C03633=1108.263,416.808,-95.419,-178.655,16.482,151.225
C03634=1108.269,417.055,-95.459,-178.654,16.489,151.227
C03635=1108.274,417.302,-95.498,-178.652,16.496,151.228
C03636=1108.279,417.549,-95.536,-178.650,16.503,151.230
C03637=1108.285,417.796,-95.575,-178.649,16.510,151.231
C03638=1108.291,418.042,-95.614,-178.647,16.517,151.232
C03639=1108.297,418.289,-95.654,-178.645,16.524,151.234
C03640=1108.302,418.536,-95.693,-178.644,16.531,151.235
C03641=1108.307,418.783,-95.733,-178.642,16.538,151.237
C03642=1108.313,419.030,-95.772,-178.640,16.545,151.238
C03643=1108.319,419.276,-95.811,-178.639,16.553,151.240
C03644=1108.325,419.523,-95.851,-178.638,16.560,151.241
C03645=1108.330,419.770,-95.890,-178.636,16.567,151.243
C03646=1108.336,420.017,-95.929,-178.634,16.574,151.244
C03647=1108.342,420.264,-95.967,-178.632,16.582,151.246
C03648=1108.347,420.510,-96.008,-178.631,16.589,151.247
C03649=1108.353,420.757,-96.047,-178.629,16.596,151.249
C03650=1108.358,421.004,-96.086,-178.627,16.603,151.250
C03651=1108.364,421.251,-96.126,-178.626,16.611,151.252
C03652=1108.370,421.497,-96.165,-178.625,16.618,151.254
C03653=1108.375,421.745,-96.205,-178.623,16.625,151.255
C03654=1108.381,421.991,-96.244,-178.621,16.633,151.257
C03655=1108.387,422.238,-96.283,-178.619,16.640,151.258
C03656=1108.392,422.485,-96.322,-178.618,16.648,151.260
C03657=1108.398,422.732,-96.362,-178.616,16.655,151.261
C03658=1108.403,422.978,-96.402,-178.615,16.663,151.263
C03659=1108.409,423.225,-96.442,-178.614,16.670,151.265
C03660=1108.414,423.443,-96.476,-178.612,16.678,151.266
C03661=1108.419,423.661,-96.511,-178.611,16.684,151.268
C03662=1108.424,423.879,-96.546,-178.610,16.691,151.269
C03663=1108.429,424.099,-96.582,-178.608,16.698,151.271
C03664=1108.434,424.317,-96.617,-178.607,16.704,151.272
C03665=1108.439,424.535,-96.652,-178.606,16.712,151.274
C03666=1108.443,424.753,-96.687,-178.604,16.718,151.275
C03667=1108.449,424.972,-96.722,-178.603,16.725,151.277
C03668=1108.454,425.218,-96.762,-178.602,16.733,151.278
C03669=1108.460,425.465,-96.802,-178.600,16.741,151.280
C03670=1108.465,425.712,-96.842,-178.599,16.749,151.282
C03671=1108.471,425.959,-96.881,-178.598,16.757,151.283
C03672=1108.477,426.205,-96.921,-178.596,16.764,151.285
C03673=1108.482,426.452,-96.961,-178.595,16.773,151.287
C03674=1108.488,426.698,-97.001,-178.593,16.781,151.289
C03675=1108.493,426.945,-97.041,-178.592,16.789,151.290
C03676=1108.500,427.192,-97.081,-178.591,16.797,151.292
C03677=1108.504,427.439,-97.121,-178.589,16.805,151.294
C03678=1108.511,427.685,-97.161,-178.588,16.813,151.296
C03679=1108.515,427.932,-97.200,-178.587,16.821,151.298
C03680=1108.522,428.178,-97.240,-178.585,16.829,151.299
C03681=1108.527,428.426,-97.281,-178.584,16.837,151.301
C03682=1108.533,428.672,-97.320,-178.583,16.845,151.303
C03683=1108.539,428.918,-97.361,-178.582,16.854,151.305
C03684=1108.544,429.165,-97.400,-178.580,16.862,151.307
C03685=1108.550,429.412,-97.441,-178.579,16.870,151.309
C03686=1108.556,429.659,-97.480,-178.578,16.879,151.311
C03687=1108.561,429.905,-97.521,-178.577,16.887,151.312
C03688=1108.566,430.152,-97.561,-178.575,16.896,151.314
C03689=1108.572,430.398,-97.601,-178.574,16.904,151.316
C03690=1108.578,430.645,-97.641,-178.573,16.913,151.318
C03691=1108.584,430.892,-97.681,-178.572,16.921,151.320
C03692=1108.589,431.138,-97.722,-178.571,16.930,151.322
C03693=1108.595,431.384,-97.762,-178.570,16.938,151.324
C03694=1108.601,431.632,-97.802,-178.568,16.946,151.326
C03695=1108.606,431.878,-97.842,-178.567,16.956,151.328
C03696=1108.611,432.125,-97.883,-178.566,16.964,151.330
C03697=1108.617,432.371,-97.924,-178.565,16.973,151.332
C03698=1108.623,432.617,-97.964,-178.564,16.981,151.334
C03699=1108.628,432.864,-98.004,-178.563,16.990,151.336
C03700=1108.634,433.111,-98.044,-178.561,16.999,151.338
C03701=1108.640,433.357,-98.084,-178.560,17.008,151.340
C03702=1108.645,433.604,-98.125,-178.560,17.017,151.342
C03703=1108.651,433.851,-98.166,-178.559,17.025,151.344
C03704=1108.656,434.097,-98.206,-178.558,17.034,151.346
C03705=1108.662,434.344,-98.247,-178.556,17.044,151.348
C03706=1108.667,434.591,-98.287,-178.556,17.052,151.351
C03707=1108.673,434.837,-98.327,-178.555,17.061,151.353
C03708=1108.679,435.083,-98.368,-178.553,17.071,151.355
C03709=1108.684,435.330,-98.409,-178.553,17.080,151.357
C03710=1108.689,435.576,-98.449,-178.552,17.089,151.359
C03711=1108.695,435.823,-98.490,-178.551,17.098,151.361
C03712=1108.701,436.069,-98.531,-178.550,17.107,151.364
C03713=1108.706,436.315,-98.572,-178.549,17.117,151.366
C03714=1108.712,436.562,-98.612,-178.549,17.126,151.368
C03715=1108.717,436.809,-98.653,-178.547,17.135,151.370
C03716=1108.723,437.037,-98.690,-178.546,17.144,151.372
C03717=1108.727,437.265,-98.728,-178.545,17.153,151.374
C03718=1108.733,437.493,-98.766,-178.545,17.161,151.376
C03719=1108.738,437.721,-98.804,-178.545,17.170,151.379
C03720=1108.743,437.949,-98.841,-178.544,17.179,151.381
C03721=1108.749,438.177,-98.879,-178.543,17.188,151.383
C03722=1108.754,438.406,-98.917,-178.542,17.196,151.385
C03723=1108.758,438.634,-98.954,-178.541,17.205,151.387
C03724=1108.764,438.880,-98.996,-178.541,17.215,151.389
C03725=1108.770,439.127,-99.037,-178.540,17.224,151.392
C03726=1108.776,439.373,-99.078,-178.539,17.234,151.394
C03727=1108.782,439.620,-99.119,-178.538,17.244,151.396
C03728=1108.787,439.866,-99.159,-178.538,17.254,151.399
C03729=1108.793,440.112,-99.201,-178.537,17.264,151.401
C03730=1108.798,440.359,-99.241,-178.536,17.273,151.403
C03731=1108.804,440.606,-99.282,-178.536,17.283,151.406
C03732=1108.810,440.852,-99.324,-178.535,17.293,151.408
C03733=1108.815,441.098,-99.364,-178.535,17.303,151.411
C03734=1108.821,441.345,-99.405,-178.534,17.313,151.413
C03735=1108.826,441.591,-99.446,-178.534,17.323,151.416
C03736=1108.832,441.838,-99.488,-178.533,17.333,151.418
C03737=1108.838,442.084,-99.530,-178.532,17.343,151.420
C03738=1108.843,442.330,-99.570,-178.532,17.353,151.423
C03739=1108.849,442.576,-99.611,-178.531,17.364,151.426
C03740=1108.854,442.823,-99.652,-178.530,17.374,151.428
C03741=1108.860,443.069,-99.694,-178.530,17.384,151.431
C03742=1108.865,443.317,-99.735,-178.530,17.394,151.433
C03743=1108.871,443.563,-99.776,-178.529,17.405,151.436
C03744=1108.876,443.808,-99.818,-178.529,17.415,151.438
C03745=1108.881,444.055,-99.859,-178.529,17.425,151.441
C03746=1108.887,444.302,-99.900,-178.529,17.435,151.444
C03747=1108.893,444.548,-99.942,-178.529,17.445,151.446
C03748=1108.899,444.795,-99.983,-178.530,17.456,151.449
C03749=1108.904,445.041,-100.025,-178.530,17.466,151.452
C03750=1108.910,445.287,-100.066,-178.530,17.477,151.454
C03751=1108.916,445.534,-100.108,-178.531,17.486,151.457
C03752=1108.921,445.781,-100.149,-178.531,17.497,151.460
C03753=1108.926,446.026,-100.190,-178.532,17.506,151.463
C03754=1108.932,446.272,-100.231,-178.533,17.517,151.465
C03755=1108.937,446.519,-100.273,-178.534,17.527,151.468
C03756=1108.943,446.766,-100.314,-178.535,17.537,151.471
C03757=1108.948,447.012,-100.356,-178.537,17.547,151.474
C03758=1108.954,447.259,-100.398,-178.538,17.557,151.477
C03759=1108.959,447.505,-100.440,-178.539,17.567,151.480
C03760=1108.965,447.751,-100.481,-178.540,17.577,151.482
C03761=1108.970,447.998,-100.523,-178.541,17.587,151.485
C03762=1108.976,448.245,-100.564,-178.544,17.597,151.488
C03763=1108.981,448.491,-100.606,-178.545,17.608,151.491
C03764=1108.987,448.737,-100.648,-178.547,17.617,151.494
C03765=1108.993,448.983,-100.689,-178.549,17.628,151.497
C03766=1108.998,449.230,-100.731,-178.551,17.637,151.500
C03767=1109.004,449.476,-100.772,-178.553,17.647,151.503
C03768=1109.010,449.723,-100.815,-178.555,17.658,151.506
C03769=1109.016,449.969,-100.856,-178.557,17.667,151.509
C03770=1109.020,450.216,-100.897,-178.559,17.677,151.512
C03771=1109.026,450.462,-100.939,-178.561,17.687,151.515
C03772=1108.617,450.455,-101.049,-178.646,17.920,151.591
C03773=1108.612,450.209,-101.007,-178.644,17.910,151.588
C03774=1108.606,449.963,-100.965,-178.642,17.900,151.585
C03775=1108.600,449.716,-100.923,-178.640,17.890,151.582
C03776=1108.594,449.470,-100.882,-178.638,17.880,151.579
C03777=1108.589,449.223,-100.840,-178.635,17.870,151.576
C03778=1108.583,448.977,-100.798,-178.634,17.859,151.573
C03779=1108.578,448.731,-100.756,-178.632,17.850,151.570
C03780=1108.572,448.484,-100.715,-178.631,17.839,151.568
C03781=1108.567,448.238,-100.673,-178.628,17.830,151.565
C03782=1108.561,447.992,-100.631,-178.627,17.819,151.562
C03783=1108.556,447.745,-100.589,-178.626,17.809,151.559
C03784=1108.550,447.498,-100.548,-178.624,17.799,151.556
C03785=1108.545,447.252,-100.506,-178.622,17.789,151.553
C03786=1108.539,447.006,-100.465,-178.621,17.779,151.550
C03787=1108.534,446.759,-100.423,-178.620,17.769,151.547
C03788=1108.528,446.513,-100.381,-178.620,17.758,151.544
C03789=1108.523,446.266,-100.339,-178.618,17.748,151.542
C03790=1108.517,446.020,-100.298,-178.617,17.738,151.539
C03791=1108.511,445.773,-100.257,-178.617,17.727,151.536
C03792=1108.506,445.528,-100.215,-178.616,17.717,151.533
C03793=1108.500,445.281,-100.174,-178.616,17.707,151.530
C03794=1108.495,445.035,-100.133,-178.615,17.696,151.528
C03795=1108.489,444.789,-100.090,-178.615,17.687,151.525
C03796=1108.484,444.542,-100.050,-178.614,17.676,151.522
C03797=1108.478,444.296,-100.008,-178.614,17.666,151.520
C03798=1108.472,444.049,-99.966,-178.614,17.656,151.517
C03799=1108.467,443.803,-99.925,-178.615,17.645,151.515
C03800=1108.461,443.556,-99.884,-178.615,17.635,151.512
C03801=1108.456,443.310,-99.842,-178.616,17.624,151.509
C03802=1108.450,443.064,-99.801,-178.616,17.614,151.507
C03803=1108.445,442.817,-99.760,-178.617,17.603,151.504
C03804=1108.439,442.571,-99.719,-178.617,17.593,151.502
C03805=1108.434,442.325,-99.677,-178.618,17.583,151.499
C03806=1108.428,442.078,-99.636,-178.618,17.573,151.497
C03807=1108.422,441.832,-99.594,-178.619,17.563,151.494
C03808=1108.417,441.585,-99.554,-178.620,17.552,151.492
C03809=1108.411,441.339,-99.513,-178.620,17.542,151.489
C03810=1108.405,441.092,-99.472,-178.621,17.532,151.487
C03811=1108.400,440.846,-99.430,-178.621,17.522,151.484
C03812=1108.394,440.600,-99.388,-178.622,17.511,151.482
C03813=1108.389,440.353,-99.348,-178.623,17.502,151.479
C03814=1108.383,440.106,-99.307,-178.624,17.492,151.477
C03815=1108.378,439.861,-99.266,-178.624,17.482,151.475
C03816=1108.372,439.614,-99.225,-178.625,17.472,151.472
C03817=1108.366,439.368,-99.184,-178.626,17.462,151.470
C03818=1108.360,439.121,-99.143,-178.626,17.453,151.467
C03819=1108.354,438.874,-99.101,-178.628,17.443,151.465
C03820=1108.349,438.628,-99.061,-178.628,17.433,151.463
C03821=1108.344,438.401,-99.023,-178.629,17.425,151.461
C03822=1108.339,438.174,-98.986,-178.630,17.416,151.459
C03823=1108.333,437.948,-98.948,-178.631,17.407,151.456
C03824=1108.328,437.721,-98.910,-178.631,17.398,151.454
C03825=1108.323,437.494,-98.873,-178.632,17.389,151.452
C03826=1108.318,437.267,-98.835,-178.633,17.380,151.450
C03827=1108.313,437.041,-98.798,-178.634,17.371,151.448
C03828=1108.308,436.815,-98.760,-178.634,17.363,151.446
C03829=1108.302,436.568,-98.719,-178.636,17.354,151.444
C03830=1108.297,436.321,-98.679,-178.636,17.344,151.442
C03831=1108.291,436.074,-98.638,-178.637,17.335,151.439
C03832=1108.286,435.828,-98.597,-178.639,17.326,151.437
C03833=1108.280,435.581,-98.557,-178.639,17.316,151.435
C03834=1108.274,435.335,-98.516,-178.640,17.308,151.433
C03835=1108.269,435.089,-98.476,-178.641,17.298,151.431
C03836=1108.263,434.843,-98.435,-178.642,17.289,151.428
C03837=1108.257,434.596,-98.394,-178.643,17.280,151.426
C03838=1108.252,434.350,-98.354,-178.644,17.270,151.424
C03839=1108.247,434.103,-98.313,-178.645,17.261,151.422
C03840=1108.241,433.856,-98.272,-178.646,17.252,151.420
C03841=1108.236,433.610,-98.232,-178.648,17.243,151.418
C03842=1108.230,433.363,-98.192,-178.649,17.234,151.416
C03843=1108.224,433.116,-98.151,-178.650,17.225,151.414
C03844=1108.218,432.870,-98.110,-178.650,17.217,151.412
C03845=1108.213,432.623,-98.070,-178.651,17.208,151.410
C03846=1108.207,432.377,-98.030,-178.653,17.198,151.408
C03847=1108.201,432.130,-97.989,-178.654,17.190,151.406
C03848=1108.196,431.883,-97.949,-178.655,17.181,151.404
C03849=1108.190,431.637,-97.909,-178.656,17.173,151.402
C03850=1108.184,431.390,-97.868,-178.657,17.164,151.400
C03851=1108.179,431.144,-97.828,-178.659,17.155,151.398
C03852=1108.173,430.897,-97.788,-178.660,17.146,151.396
C03853=1108.167,430.651,-97.747,-178.661,17.138,151.394
C03854=1108.163,430.404,-97.707,-178.662,17.129,151.392
C03855=1108.156,430.157,-97.667,-178.663,17.121,151.390
C03856=1108.151,429.911,-97.627,-178.665,17.113,151.388
C03857=1108.146,429.664,-97.587,-178.667,17.104,151.386
C03858=1108.139,429.417,-97.547,-178.668,17.095,151.384
C03859=1108.134,429.171,-97.506,-178.669,17.087,151.382
C03860=1108.128,428.925,-97.466,-178.670,17.078,151.380
C03861=1108.123,428.677,-97.426,-178.671,17.070,151.378
C03862=1108.118,428.431,-97.386,-178.673,17.062,151.377
C03863=1108.112,428.184,-97.346,-178.674,17.054,151.375
C03864=1108.106,427.937,-97.306,-178.675,17.046,151.373
C03865=1108.100,427.691,-97.266,-178.677,17.037,151.371
C03866=1108.095,427.444,-97.226,-178.678,17.029,151.369
C03867=1108.089,427.198,-97.186,-178.679,17.021,151.367
C03868=1108.083,426.951,-97.147,-178.681,17.013,151.366
C03869=1108.077,426.704,-97.106,-178.682,17.005,151.364
C03870=1108.072,426.458,-97.067,-178.684,16.997,151.362
C03871=1108.066,426.211,-97.026,-178.685,16.989,151.360
C03872=1108.061,425.964,-96.987,-178.686,16.981,151.359
C03873=1108.055,425.718,-96.946,-178.688,16.973,151.357
C03874=1108.050,425.471,-96.907,-178.689,16.965,151.355
C03875=1108.044,425.224,-96.867,-178.691,16.957,151.353
C03876=1108.039,424.978,-96.827,-178.692,16.949,151.352
C03877=1108.033,424.759,-96.793,-178.693,16.942,151.350
C03878=1108.029,424.540,-96.757,-178.695,16.935,151.349
C03879=1108.023,424.322,-96.721,-178.696,16.928,151.347
C03880=1108.019,424.103,-96.687,-178.697,16.921,151.346
C03881=1108.013,423.885,-96.652,-178.699,16.914,151.344
C03882=1108.009,423.666,-96.616,-178.700,16.907,151.343
C03883=1108.004,423.448,-96.581,-178.702,16.901,151.341
C03884=1107.999,423.230,-96.546,-178.703,16.894,151.340
C03885=1107.993,422.983,-96.506,-178.704,16.886,151.338
C03886=1107.988,422.736,-96.467,-178.706,16.878,151.336
C03887=1107.982,422.489,-96.427,-178.708,16.871,151.335
C03888=1107.976,422.243,-96.387,-178.709,16.863,151.333
C03889=1107.970,421.996,-96.348,-178.711,16.855,151.332
C03890=1107.965,421.750,-96.309,-178.712,16.848,151.330
C03891=1107.959,421.502,-96.269,-178.714,16.841,151.329
C03892=1107.954,421.256,-96.230,-178.715,16.833,151.327
C03893=1107.948,421.009,-96.190,-178.717,16.826,151.325
C03894=1107.942,420.762,-96.151,-178.719,16.818,151.324
C03895=1107.936,420.515,-96.112,-178.720,16.811,151.322
C03896=1107.931,420.268,-96.072,-178.722,16.804,151.321
C03897=1107.925,420.021,-96.033,-178.724,16.796,151.319
C03898=1107.920,419.775,-95.993,-178.725,16.789,151.318
C03899=1107.914,419.528,-95.954,-178.727,16.782,151.316
C03900=1107.908,419.282,-95.915,-178.728,16.775,151.315
C03901=1107.902,419.034,-95.876,-178.730,16.767,151.313
C03902=1107.898,418.787,-95.836,-178.732,16.760,151.312
C03903=1107.891,418.540,-95.797,-178.734,16.753,151.310
C03904=1107.886,418.294,-95.758,-178.735,16.746,151.309
C03905=1107.881,418.047,-95.719,-178.737,16.738,151.307
C03906=1107.874,417.800,-95.679,-178.739,16.731,151.306
C03907=1107.869,417.554,-95.640,-178.740,16.725,151.304
C03908=1107.863,417.307,-95.601,-178.742,16.717,151.303
C03909=1107.857,417.060,-95.562,-178.744,16.710,151.302
C03910=1107.853,416.813,-95.523,-178.746,16.703,151.300
C03911=1107.847,416.566,-95.483,-178.747,16.696,151.299
C03912=1107.841,416.320,-95.445,-178.749,16.689,151.297
C03913=1107.835,416.072,-95.405,-178.751,16.683,151.296
C03914=1107.829,415.826,-95.366,-178.753,16.676,151.294
C03915=1107.823,415.578,-95.328,-178.755,16.669,151.293
C03916=1107.818,415.332,-95.288,-178.756,16.662,151.292
C03917=1107.812,415.085,-95.249,-178.758,16.655,151.290
C03918=1107.807,414.838,-95.211,-178.760,16.649,151.289
C03919=1107.801,414.591,-95.172,-178.762,16.642,151.288
C03920=1107.795,414.344,-95.132,-178.764,16.635,151.286
C03921=1107.790,414.097,-95.094,-178.765,16.628,151.285
C03922=1107.785,413.851,-95.055,-178.768,16.621,151.284
C03923=1107.778,413.604,-95.016,-178.769,16.615,151.282
C03924=1107.773,413.357,-94.978,-178.771,16.608,151.281
C03925=1107.767,413.110,-94.939,-178.773,16.602,151.280
C03926=1107.761,412.863,-94.900,-178.775,16.595,151.279
C03927=1107.756,412.616,-94.861,-178.776,16.589,151.277
C03928=1107.751,412.369,-94.822,-178.779,16.582,151.276
C03929=1107.745,412.122,-94.783,-178.780,16.576,151.275
C03930=1107.739,411.875,-94.745,-178.782,16.569,151.273
C03931=1107.733,411.629,-94.706,-178.784,16.563,151.272
C03932=1107.727,411.381,-94.667,-178.786,16.556,151.271
C03933=1107.723,411.169,-94.634,-178.788,16.550,151.270
C03934=1107.717,410.957,-94.601,-178.789,16.545,151.269
C03935=1107.713,410.746,-94.568,-178.791,16.539,151.268
C03936=1107.708,410.534,-94.535,-178.793,16.534,151.267
C03937=1107.703,410.322,-94.502,-178.794,16.529,151.266
C03938=1107.699,410.109,-94.469,-178.796,16.523,151.265
C03939=1107.694,409.897,-94.436,-178.798,16.517,151.264
C03940=1107.689,409.686,-94.402,-178.799,16.512,151.263
C03941=1107.683,409.439,-94.364,-178.802,16.506,151.261
C03942=1107.677,409.191,-94.325,-178.803,16.500,151.260
C03943=1107.672,408.945,-94.286,-178.805,16.494,151.259
C03944=1107.667,408.698,-94.248,-178.807,16.487,151.258
C03945=1107.661,408.451,-94.210,-178.809,16.481,151.257
C03946=1107.656,408.204,-94.172,-178.811,16.474,151.256
C03947=1107.650,407.956,-94.133,-178.813,16.468,151.254
C03948=1107.644,407.710,-94.095,-178.815,16.463,151.253
C03949=1107.639,407.463,-94.056,-178.817,16.456,151.252
C03950=1107.633,407.216,-94.018,-178.819,16.450,151.251
C03951=1107.627,406.968,-93.980,-178.821,16.444,151.250
C03952=1107.622,406.721,-93.941,-178.823,16.438,151.249
C03953=1107.616,406.475,-93.902,-178.825,16.432,151.248
C03954=1107.610,406.228,-93.865,-178.827,16.426,151.247
C03955=1107.605,405.981,-93.826,-178.829,16.420,151.245
C03956=1107.599,405.734,-93.788,-178.831,16.414,151.244
C03957=1107.594,405.487,-93.750,-178.833,16.408,151.243
C03958=1107.588,405.240,-93.712,-178.835,16.402,151.242
C03959=1107.582,404.993,-93.674,-178.838,16.396,151.241
C03960=1107.577,404.746,-93.636,-178.839,16.391,151.240
C03961=1107.571,404.498,-93.597,-178.841,16.385,151.239
C03962=1107.565,404.252,-93.559,-178.843,16.379,151.238
C03963=1107.560,404.005,-93.521,-178.846,16.373,151.237
C03964=1107.554,403.758,-93.483,-178.848,16.367,151.236
C03965=1107.549,403.511,-93.445,-178.850,16.362,151.235
C03966=1107.542,403.263,-93.407,-178.852,16.356,151.234
C03967=1107.536,403.017,-93.369,-178.854,16.351,151.233
C03968=1107.531,402.769,-93.331,-178.856,16.345,151.232
C03969=1107.525,402.523,-93.293,-178.859,16.339,151.231
C03970=1107.520,402.275,-93.255,-178.860,16.333,151.230
C03971=1107.514,402.028,-93.218,-178.863,16.328,151.229
C03972=1107.509,401.782,-93.180,-178.865,16.322,151.228
C03973=1107.503,401.535,-93.142,-178.867,16.317,151.227
C03974=1107.497,401.287,-93.103,-178.869,16.311,151.226
C03975=1107.492,401.040,-93.065,-178.871,16.305,151.225
C03976=1107.486,400.793,-93.028,-178.874,16.300,151.224
C03977=1107.480,400.546,-92.990,-178.876,16.294,151.223
C03978=1107.475,400.299,-92.952,-178.878,16.289,151.223
C03979=1107.469,400.052,-92.914,-178.880,16.284,151.222
C03980=1107.464,399.805,-92.877,-178.882,16.278,151.221
C03981=1107.458,399.558,-92.839,-178.884,16.273,151.220
C03982=1107.452,399.311,-92.801,-178.886,16.267,151.219
C03983=1107.447,399.064,-92.764,-178.888,16.262,151.218
C03984=1107.441,398.817,-92.726,-178.890,16.257,151.217
C03985=1107.435,398.570,-92.688,-178.893,16.251,151.216
C03986=1107.430,398.322,-92.651,-178.895,16.246,151.215
C03987=1107.424,398.076,-92.613,-178.897,16.241,151.214
C03988=1107.418,397.829,-92.575,-178.899,16.235,151.214
C03989=1107.414,397.616,-92.543,-178.902,16.231,151.213
C03990=1107.408,397.404,-92.511,-178.903,16.226,151.212
C03991=1107.404,397.192,-92.478,-178.905,16.222,151.211
C03992=1107.398,396.979,-92.447,-178.907,16.217,151.211
C03993=1107.394,396.768,-92.414,-178.909,16.213,151.210
C03994=1107.389,396.555,-92.382,-178.911,16.208,151.209
C03995=1107.384,396.343,-92.350,-178.913,16.204,151.209
C03996=1107.380,396.131,-92.317,-178.915,16.199,151.208
C03997=1107.374,395.884,-92.280,-178.917,16.194,151.207
C03998=1107.368,395.637,-92.243,-178.920,16.189,151.206
C03999=1107.363,395.390,-92.206,-178.922,16.184,151.205
C04000=1107.357,395.143,-92.168,-178.924,16.179,151.205
C04001=1107.351,394.896,-92.131,-178.927,16.174,151.204
C04002=1107.346,394.648,-92.094,-178.929,16.168,151.203
C04003=1107.340,394.401,-92.056,-178.931,16.164,151.202
C04004=1107.334,394.154,-92.019,-178.934,16.159,151.202
C04005=1107.328,393.907,-91.981,-178.936,16.153,151.201
C04006=1107.323,393.660,-91.944,-178.938,16.149,151.200
C04007=1107.317,393.413,-91.907,-178.940,16.144,151.199
C04008=1107.311,393.166,-91.869,-178.943,16.139,151.198
C04009=1107.306,392.919,-91.832,-178.945,16.134,151.198
C04010=1107.300,392.671,-91.795,-178.948,16.129,151.197
C04011=1107.294,392.424,-91.758,-178.950,16.124,151.196
C04012=1107.289,392.178,-91.721,-178.953,16.119,151.196
C04013=1107.283,391.930,-91.684,-178.955,16.115,151.195
C04014=1107.278,391.683,-91.647,-178.958,16.110,151.194
C04015=1107.272,391.436,-91.610,-178.960,16.105,151.193
C04016=1107.266,391.189,-91.573,-178.962,16.101,151.193
C04017=1107.260,390.942,-91.536,-178.964,16.096,151.192
C04018=1107.254,390.695,-91.499,-178.967,16.091,151.191
C04019=1107.249,390.447,-91.462,-178.969,16.086,151.191
C04020=1107.243,390.200,-91.424,-178.972,16.081,151.190
C04021=1107.238,389.954,-91.387,-178.975,16.076,151.189
C04022=1107.232,389.707,-91.351,-178.977,16.072,151.189
C04023=1107.226,389.459,-91.314,-178.979,16.067,151.188
C04024=1107.220,389.212,-91.277,-178.981,16.062,151.187
C04025=1107.215,388.965,-91.240,-178.984,16.058,151.187
C04026=1107.208,388.718,-91.203,-178.987,16.053,151.186
C04027=1107.203,388.471,-91.166,-178.989,16.048,151.186
C04028=1107.198,388.224,-91.129,-178.992,16.044,151.185
C04029=1107.192,387.976,-91.092,-178.994,16.040,151.184
C04030=1107.186,387.729,-91.056,-178.996,16.035,151.184
C04031=1107.180,387.482,-91.019,-178.999,16.030,151.183
C04032=1107.175,387.235,-90.982,-179.002,16.025,151.182
C04033=1107.170,386.988,-90.945,-179.004,16.021,151.182
C04034=1107.163,386.741,-90.909,-179.007,16.016,151.181
C04035=1107.158,386.493,-90.872,-179.009,16.012,151.181
C04036=1107.153,386.247,-90.835,-179.012,16.008,151.180
C04037=1107.146,386.000,-90.799,-179.014,16.003,151.179
C04038=1107.141,385.752,-90.761,-179.017,15.998,151.179
C04039=1107.136,385.506,-90.725,-179.019,15.994,151.178
C04040=1107.130,385.259,-90.688,-179.022,15.990,151.178
C04041=1107.124,385.011,-90.652,-179.024,15.985,151.177
C04042=1107.119,384.763,-90.615,-179.027,15.980,151.176
C04043=1107.113,384.517,-90.579,-179.029,15.977,151.176
C04044=1107.107,384.269,-90.542,-179.032,15.972,151.175
C04045=1107.098,383.857,-90.481,-179.036,15.965,151.175
C04046=1107.089,383.444,-90.420,-179.041,15.957,151.174
C04047=1107.080,383.032,-90.359,-179.045,15.950,151.173
C04048=1107.070,382.620,-90.298,-179.049,15.943,151.172
C04049=1107.064,382.373,-90.263,-179.052,15.939,151.171
C04050=1107.059,382.126,-90.226,-179.055,15.935,151.171
C04051=1107.052,381.879,-90.189,-179.057,15.930,151.170
C04052=1107.048,381.631,-90.153,-179.060,15.926,151.170
C04053=1107.041,381.384,-90.117,-179.063,15.922,151.169
C04054=1107.036,381.136,-90.080,-179.065,15.918,151.169
C04055=1107.030,380.889,-90.044,-179.068,15.913,151.168
C04056=1107.024,380.643,-90.008,-179.070,15.910,151.168
C04057=1107.019,380.395,-89.972,-179.073,15.905,151.167
C04058=1107.012,380.148,-89.935,-179.076,15.902,151.167
C04059=1107.008,379.901,-89.899,-179.078,15.897,151.167
C04060=1107.001,379.653,-89.863,-179.081,15.893,151.166
C04061=1106.996,379.407,-89.827,-179.083,15.889,151.166
C04062=1106.990,379.159,-89.790,-179.087,15.885,151.165
C04063=1106.984,378.911,-89.755,-179.089,15.881,151.165
C04064=1106.978,378.665,-89.719,-179.092,15.877,151.164
C04065=1106.973,378.417,-89.682,-179.095,15.873,151.164
C04066=1106.967,378.169,-89.647,-179.098,15.868,151.163
C04067=1106.962,377.923,-89.610,-179.100,15.865,151.163
C04068=1106.956,377.675,-89.574,-179.103,15.861,151.163
C04069=1106.950,377.429,-89.538,-179.105,15.857,151.162
C04070=1106.945,377.181,-89.502,-179.108,15.853,151.162
C04071=1106.940,376.934,-89.466,-179.111,15.849,151.161
C04072=1106.933,376.687,-89.430,-179.113,15.845,151.161
C04073=1106.928,376.439,-89.394,-179.117,15.841,151.161
C04074=1106.923,376.192,-89.358,-179.119,15.838,151.160
C04075=1106.916,375.945,-89.322,-179.122,15.833,151.160
C04076=1106.911,375.698,-89.286,-179.124,15.830,151.159
C04077=1106.906,375.450,-89.250,-179.127,15.825,151.159
C04078=1106.900,375.203,-89.215,-179.130,15.821,151.159
C04079=1106.894,374.955,-89.179,-179.132,15.818,151.158
C04080=1106.888,374.709,-89.143,-179.136,15.814,151.158
C04081=1106.883,374.461,-89.107,-179.138,15.810,151.158
C04082=1106.878,374.214,-89.071,-179.141,15.806,151.157
C04083=1106.872,373.966,-89.035,-179.144,15.803,151.157
C04084=1106.866,373.718,-89.000,-179.147,15.799,151.157
C04085=1106.860,373.472,-88.964,-179.149,15.795,151.156
C04086=1106.854,373.224,-88.928,-179.152,15.792,151.156
C04087=1106.848,372.977,-88.893,-179.155,15.788,151.156
C04088=1106.842,372.730,-88.857,-179.158,15.784,151.155
C04089=1106.838,372.483,-88.821,-179.161,15.781,151.155
C04090=1106.832,372.235,-88.785,-179.164,15.777,151.155
C04091=1106.826,371.988,-88.750,-179.166,15.773,151.154
C04092=1106.820,371.740,-88.714,-179.169,15.769,151.154
C04093=1106.815,371.493,-88.679,-179.172,15.766,151.154
C04094=1106.809,371.246,-88.643,-179.175,15.762,151.154
C04095=1106.803,370.999,-88.608,-179.177,15.759,151.153
C04096=1106.797,370.751,-88.572,-179.181,15.755,151.153
C04097=1106.788,370.365,-88.517,-179.185,15.749,151.152
C04098=1106.779,369.980,-88.461,-179.190,15.744,151.152
C04099=1106.770,369.594,-88.406,-179.194,15.738,151.152
C04100=1106.762,369.208,-88.351,-179.199,15.733,151.151
C04101=1106.757,368.961,-88.315,-179.201,15.729,151.151
C04102=1106.751,368.714,-88.280,-179.204,15.725,151.151
C04103=1106.746,368.467,-88.244,-179.207,15.722,151.150
C04104=1106.739,368.219,-88.210,-179.209,15.719,151.150
C04105=1106.734,367.972,-88.174,-179.213,15.715,151.150
C04106=1106.728,367.725,-88.139,-179.215,15.712,151.150
C04107=1106.722,367.477,-88.103,-179.219,15.708,151.149
C04108=1106.717,367.229,-88.069,-179.221,15.705,151.149
C04109=1106.711,366.982,-88.033,-179.225,15.701,151.149
C04110=1106.706,366.735,-87.998,-179.227,15.698,151.149
C04111=1106.700,366.488,-87.962,-179.230,15.695,151.148
C04112=1106.694,366.239,-87.927,-179.233,15.691,151.148
C04113=1106.689,365.993,-87.892,-179.236,15.688,151.148
C04114=1106.683,365.744,-87.857,-179.239,15.684,151.148
C04115=1106.678,365.497,-87.821,-179.242,15.681,151.148
C04116=1106.672,365.251,-87.787,-179.244,15.678,151.147
C04117=1106.666,365.002,-87.752,-179.248,15.674,151.147
C04118=1106.661,364.755,-87.716,-179.251,15.671,151.147
C04119=1106.655,364.508,-87.681,-179.253,15.668,151.147
C04120=1106.649,364.260,-87.646,-179.257,15.664,151.147
C04121=1106.643,364.013,-87.611,-179.259,15.661,151.146
C04122=1106.637,363.765,-87.576,-179.263,15.658,151.146
C04123=1106.632,363.518,-87.541,-179.266,15.655,151.146
C04124=1106.627,363.271,-87.506,-179.268,15.652,151.146
C04125=1106.620,363.023,-87.471,-179.272,15.648,151.146
C04126=1106.615,362.776,-87.436,-179.275,15.645,151.146
C04127=1106.610,362.529,-87.401,-179.277,15.642,151.146
C04128=1106.603,362.281,-87.367,-179.281,15.638,151.145
C04129=1106.598,362.033,-87.332,-179.284,15.635,151.145
C04130=1106.593,361.786,-87.297,-179.286,15.632,151.145
C04131=1106.586,361.538,-87.262,-179.290,15.629,151.145
C04132=1106.581,361.291,-87.227,-179.292,15.626,151.145
C04133=1106.576,361.043,-87.192,-179.295,15.623,151.145
C04134=1106.569,360.795,-87.158,-179.299,15.619,151.145
C04135=1106.564,360.549,-87.122,-179.301,15.616,151.144
C04136=1106.559,360.301,-87.088,-179.304,15.613,151.144
C04137=1106.553,360.054,-87.054,-179.308,15.610,151.144
C04138=1106.547,359.806,-87.018,-179.311,15.607,151.144
C04139=1106.542,359.558,-86.983,-179.313,15.604,151.144
C04140=1106.536,359.311,-86.949,-179.316,15.601,151.144
C04141=1106.530,359.063,-86.914,-179.320,15.598,151.144
C04142=1106.524,358.816,-86.879,-179.323,15.595,151.144
C04143=1106.519,358.569,-86.845,-179.326,15.592,151.144
C04144=1106.512,358.321,-86.810,-179.329,15.588,151.143
C04145=1106.507,358.073,-86.776,-179.332,15.586,151.143
C04146=1106.501,357.826,-86.742,-179.335,15.583,151.143
C04147=1106.496,357.579,-86.706,-179.338,15.580,151.143
C04148=1106.489,357.331,-86.672,-179.341,15.577,151.143
C04149=1106.481,356.960,-86.620,-179.346,15.572,151.143
C04150=1106.472,356.589,-86.568,-179.350,15.568,151.143
C04151=1106.464,356.218,-86.517,-179.355,15.563,151.143
C04152=1106.457,355.847,-86.465,-179.359,15.559,151.143
C04153=1106.450,355.599,-86.431,-179.362,15.557,151.143
C04154=1106.444,355.352,-86.397,-179.366,15.553,151.143
C04155=1106.439,355.105,-86.362,-179.369,15.550,151.143
C04156=1106.433,354.857,-86.328,-179.372,15.548,151.143
C04157=1106.428,354.610,-86.294,-179.375,15.545,151.143
C04158=1106.422,354.362,-86.259,-179.378,15.542,151.143
C04159=1106.417,354.114,-86.224,-179.382,15.539,151.143
C04160=1106.411,353.867,-86.190,-179.385,15.536,151.143
C04161=1106.405,353.620,-86.156,-179.388,15.534,151.142
C04162=1106.400,353.372,-86.122,-179.390,15.531,151.142
C04163=1106.394,353.125,-86.088,-179.393,15.528,151.142
C04164=1106.388,352.877,-86.053,-179.397,15.525,151.142
C04165=1106.382,352.629,-86.019,-179.400,15.522,151.142
C04166=1106.377,352.381,-85.985,-179.403,15.519,151.142
C04167=1106.371,352.134,-85.951,-179.406,15.517,151.142
C04168=1106.366,351.886,-85.917,-179.409,15.514,151.142
C04169=1106.360,351.639,-85.883,-179.413,15.511,151.142
C04170=1106.354,351.391,-85.848,-179.416,15.508,151.142
C04171=1106.348,351.143,-85.815,-179.419,15.506,151.142
C04172=1106.343,350.896,-85.780,-179.422,15.503,151.142
C04173=1106.337,350.648,-85.746,-179.425,15.501,151.142
C04174=1106.331,350.401,-85.712,-179.428,15.498,151.142
C04175=1106.326,350.153,-85.679,-179.432,15.495,151.143
C04176=1106.320,349.905,-85.644,-179.435,15.492,151.143
C04177=1106.315,349.658,-85.610,-179.438,15.489,151.142
C04178=1106.308,349.410,-85.576,-179.441,15.487,151.143
C04179=1106.303,349.162,-85.542,-179.444,15.484,151.143
C04180=1106.297,348.915,-85.508,-179.447,15.482,151.143
C04181=1106.292,348.667,-85.474,-179.450,15.479,151.143
C04182=1106.286,348.420,-85.440,-179.454,15.476,151.143
C04183=1106.280,348.172,-85.407,-179.457,15.474,151.143
C04184=1106.275,347.924,-85.373,-179.460,15.471,151.143
C04185=1106.269,347.677,-85.339,-179.464,15.469,151.143
C04186=1106.263,347.429,-85.305,-179.467,15.466,151.143
C04187=1106.257,347.182,-85.271,-179.470,15.464,151.143
C04188=1106.253,346.934,-85.237,-179.473,15.461,151.143
C04189=1106.247,346.686,-85.203,-179.476,15.459,151.143
C04190=1106.241,346.438,-85.170,-179.480,15.455,151.143
C04191=1106.235,346.191,-85.136,-179.483,15.453,151.143
C04192=1106.230,345.943,-85.103,-179.486,15.451,151.143
C04193=1106.224,345.696,-85.069,-179.489,15.448,151.143
C04194=1106.218,345.448,-85.035,-179.492,15.446,151.144
C04195=1106.213,345.200,-85.002,-179.496,15.443,151.144
C04196=1106.206,344.952,-84.967,-179.499,15.441,151.144
C04197=1106.201,344.704,-84.934,-179.502,15.438,151.144
C04198=1106.195,344.457,-84.900,-179.505,15.436,151.144
C04199=1106.189,344.209,-84.867,-179.509,15.434,151.144
C04200=1106.184,343.961,-84.833,-179.511,15.431,151.144
C04201=1106.176,343.593,-84.784,-179.517,15.428,151.144
C04202=1106.167,343.224,-84.734,-179.521,15.424,151.144
C04203=1106.158,342.856,-84.684,-179.526,15.420,151.145
C04204=1106.150,342.487,-84.634,-179.531,15.417,151.145
C04205=1106.144,342.239,-84.601,-179.535,15.414,151.145
C04206=1106.139,341.991,-84.567,-179.538,15.411,151.145
C04207=1106.133,341.744,-84.533,-179.541,15.409,151.145
C04208=1106.127,341.496,-84.500,-179.545,15.407,151.145
C04209=1106.122,341.248,-84.467,-179.548,15.404,151.145
C04210=1106.117,341.001,-84.434,-179.551,15.402,151.146
C04211=1106.110,340.753,-84.401,-179.554,15.400,151.146
C04212=1106.104,340.506,-84.367,-179.558,15.398,151.146
C04213=1106.099,340.258,-84.333,-179.561,15.395,151.146
C04214=1106.093,340.010,-84.300,-179.564,15.393,151.146
C04215=1106.088,339.762,-84.267,-179.568,15.391,151.146
C04216=1106.082,339.514,-84.233,-179.571,15.388,151.146
C04217=1106.076,339.267,-84.201,-179.574,15.386,151.147
C04218=1106.070,339.019,-84.167,-179.577,15.384,151.147
C04219=1106.065,338.771,-84.134,-179.581,15.381,151.147
C04220=1106.059,338.523,-84.101,-179.584,15.379,151.147
C04221=1106.054,338.276,-84.068,-179.587,15.377,151.147
C04222=1106.048,338.028,-84.035,-179.591,15.375,151.147
C04223=1106.042,337.780,-84.002,-179.594,15.373,151.148
C04224=1106.037,337.532,-83.968,-179.597,15.370,151.148
C04225=1106.031,337.285,-83.936,-179.601,15.368,151.148
C04226=1106.025,337.037,-83.902,-179.604,15.366,151.148
C04227=1106.020,336.789,-83.869,-179.607,15.364,151.148
C04228=1106.013,336.541,-83.836,-179.611,15.361,151.148
C04229=1106.008,336.293,-83.803,-179.614,15.360,151.149
C04230=1106.003,336.046,-83.770,-179.617,15.358,151.149
C04231=1105.996,335.799,-83.737,-179.620,15.356,151.149
C04232=1105.991,335.550,-83.704,-179.623,15.353,151.149
C04233=1105.986,335.302,-83.671,-179.627,15.351,151.150
C04234=1105.979,335.055,-83.638,-179.630,15.349,151.150
C04235=1105.974,334.807,-83.605,-179.634,15.347,151.150
C04236=1105.969,334.559,-83.572,-179.637,15.345,151.150
C04237=1105.963,334.311,-83.540,-179.640,15.342,151.150
C04238=1105.957,334.063,-83.507,-179.644,15.341,151.151
C04239=1105.951,333.816,-83.474,-179.647,15.338,151.151
C04240=1105.945,333.568,-83.441,-179.651,15.336,151.151
C04241=1105.941,333.320,-83.408,-179.654,15.334,151.151
C04242=1105.935,333.072,-83.376,-179.657,15.332,151.151
C04243=1105.929,332.824,-83.342,-179.661,15.330,151.152
C04244=1105.923,332.576,-83.310,-179.664,15.328,151.152
C04245=1105.918,332.329,-83.277,-179.667,15.326,151.152
C04246=1105.912,332.081,-83.245,-179.670,15.324,151.152
C04247=1105.906,331.833,-83.212,-179.674,15.322,151.153
C04248=1105.900,331.585,-83.179,-179.678,15.320,151.153
C04249=1105.895,331.337,-83.146,-179.681,15.318,151.153
C04250=1105.889,331.089,-83.114,-179.684,15.316,151.153
C04251=1105.883,330.842,-83.081,-179.688,15.314,151.154
C04252=1105.877,330.594,-83.048,-179.691,15.312,151.154
C04253=1105.869,330.219,-83.000,-179.696,15.310,151.154
C04254=1105.860,329.845,-82.950,-179.701,15.307,151.155
C04255=1105.851,329.470,-82.901,-179.706,15.303,151.155
C04256=1105.842,329.095,-82.852,-179.712,15.301,151.156
C04257=1105.837,328.847,-82.819,-179.715,15.299,151.156
C04258=1105.831,328.599,-82.787,-179.719,15.297,151.156
C04259=1105.825,328.351,-82.754,-179.722,15.295,151.156
C04260=1105.820,328.103,-82.722,-179.725,15.293,151.157
C04261=1105.814,327.856,-82.689,-179.729,15.291,151.157
C04262=1105.808,327.608,-82.657,-179.732,15.289,151.157
C04263=1105.802,327.360,-82.626,-179.736,15.288,151.158
C04264=1105.797,327.112,-82.592,-179.740,15.286,151.158
C04265=1105.791,326.864,-82.560,-179.742,15.284,151.158
C04266=1105.785,326.616,-82.528,-179.746,15.282,151.158
C04267=1105.779,326.369,-82.496,-179.749,15.280,151.159
C04268=1105.774,326.120,-82.463,-179.753,15.278,151.159
C04269=1105.768,325.872,-82.431,-179.756,15.276,151.159
C04270=1105.762,325.625,-82.399,-179.760,15.274,151.160
C04271=1105.756,325.377,-82.367,-179.763,15.273,151.160
C04272=1105.751,325.129,-82.334,-179.766,15.271,151.160
C04273=1105.745,324.882,-82.302,-179.770,15.269,151.161
C04274=1105.739,324.633,-82.270,-179.774,15.268,151.161
C04275=1105.734,324.386,-82.238,-179.777,15.266,151.161
C04276=1105.728,324.138,-82.206,-179.780,15.264,151.162
C04277=1105.723,323.889,-82.173,-179.783,15.262,151.162
C04278=1105.717,323.642,-82.141,-179.787,15.260,151.162
C04279=1105.711,323.394,-82.109,-179.791,15.258,151.162
C04280=1105.705,323.147,-82.077,-179.794,15.256,151.163
C04281=1105.699,322.898,-82.045,-179.797,15.255,151.163
C04282=1105.693,322.650,-82.013,-179.801,15.254,151.164
C04283=1105.689,322.402,-81.981,-179.805,15.252,151.164
C04284=1105.683,322.154,-81.949,-179.808,15.250,151.164
C04285=1105.677,321.907,-81.917,-179.811,15.249,151.164
C04286=1105.671,321.659,-81.885,-179.815,15.247,151.165
C04287=1105.666,321.412,-81.853,-179.818,15.245,151.165
C04288=1105.660,321.163,-81.821,-179.822,15.243,151.165
C04289=1105.654,320.916,-81.789,-179.825,15.241,151.166
C04290=1105.648,320.668,-81.757,-179.828,15.240,151.166
C04291=1105.643,320.420,-81.726,-179.832,15.238,151.166
C04292=1105.638,320.172,-81.693,-179.835,15.236,151.167
C04293=1105.632,319.924,-81.661,-179.839,15.234,151.167
C04294=1105.626,319.676,-81.629,-179.842,15.233,151.167
C04295=1105.621,319.428,-81.598,-179.846,15.231,151.168
C04296=1105.615,319.179,-81.566,-179.849,15.229,151.168
C04297=1105.610,318.932,-81.535,-179.853,15.228,151.169
C04298=1105.604,318.684,-81.503,-179.856,15.226,151.169
C04299=1105.599,318.436,-81.471,-179.860,15.224,151.169
C04300=1105.593,318.188,-81.439,-179.863,15.223,151.169
C04301=1105.587,317.941,-81.407,-179.867,15.221,151.170
C04302=1105.581,317.692,-81.375,-179.870,15.220,151.170
C04303=1105.576,317.445,-81.343,-179.873,15.218,151.171
C04304=1105.571,317.197,-81.313,-179.877,15.216,151.171
C04305=1105.562,316.815,-81.264,-179.883,15.214,151.172
C04306=1105.554,316.433,-81.214,-179.887,15.211,151.172
C04307=1105.545,316.051,-81.166,-179.893,15.209,151.173
C04308=1105.536,315.669,-81.117,-179.899,15.206,151.173
C04309=1105.531,315.421,-81.085,-179.902,15.204,151.174
C04310=1105.525,315.173,-81.054,-179.905,15.203,151.174
C04311=1105.519,314.925,-81.023,-179.909,15.202,151.174
C04312=1105.513,314.678,-80.991,-179.913,15.200,151.175
C04313=1105.508,314.429,-80.960,-179.916,15.199,151.175
C04314=1105.502,314.181,-80.928,-179.920,15.197,151.176
C04315=1105.496,313.934,-80.897,-179.924,15.196,151.176
C04316=1105.491,313.685,-80.866,-179.926,15.195,151.177
C04317=1105.485,313.437,-80.834,-179.930,15.193,151.177
C04318=1105.478,313.190,-80.803,-179.934,15.191,151.177
C04319=1105.473,312.941,-80.771,-179.937,15.190,151.178
C04320=1105.467,312.694,-80.740,-179.941,15.189,151.178
C04321=1105.462,312.446,-80.709,-179.945,15.187,151.179
C04322=1105.456,312.198,-80.677,-179.948,15.186,151.179
C04323=1105.450,311.950,-80.646,-179.951,15.184,151.179
C04324=1105.444,311.702,-80.615,-179.955,15.183,151.180
C04325=1105.438,311.454,-80.583,-179.959,15.182,151.180
C04326=1105.433,311.206,-80.553,-179.962,15.180,151.181
C04327=1105.427,310.958,-80.521,-179.966,15.179,151.181
C04328=1105.421,310.710,-80.490,-179.969,15.178,151.182
C04329=1105.415,310.463,-80.459,-179.973,15.176,151.182
C04330=1105.410,310.214,-80.428,-179.977,15.174,151.183
C04331=1105.404,309.967,-80.397,-179.980,15.174,151.183
C04332=1105.398,309.719,-80.366,-179.984,15.172,151.183
C04333=1105.393,309.470,-80.334,-179.988,15.170,151.184
C04334=1105.387,309.223,-80.303,-179.991,15.169,151.184
C04335=1105.382,308.974,-80.272,-179.994,15.168,151.185
C04336=1105.375,308.726,-80.241,-179.998,15.166,151.185
C04337=1105.370,308.478,-80.210,179.999,15.165,151.186
C04338=1105.364,308.231,-80.180,179.995,15.164,151.186
C04339=1105.359,307.983,-80.148,179.992,15.163,151.187
C04340=1105.352,307.734,-80.117,179.988,15.161,151.187
C04341=1105.347,307.486,-80.086,179.984,15.160,151.188
C04342=1105.342,307.239,-80.055,179.981,15.159,151.188
C04343=1105.336,306.991,-80.024,179.977,15.157,151.188
C04344=1105.329,306.742,-79.994,179.973,15.155,151.189
C04345=1105.324,306.494,-79.963,179.970,15.155,151.189
C04346=1105.318,306.247,-79.932,179.966,15.153,151.190
C04347=1105.313,305.999,-79.901,179.962,15.152,151.190
C04348=1105.307,305.751,-79.870,179.959,15.150,151.191
C04349=1105.302,305.502,-79.839,179.955,15.149,151.191
C04350=1105.296,305.255,-79.809,179.951,15.147,151.192
C04351=1105.290,305.007,-79.777,179.948,15.147,151.192
C04352=1105.285,304.759,-79.747,179.944,15.145,151.193
C04353=1105.280,304.511,-79.716,179.941,15.144,151.193
C04354=1105.273,304.263,-79.685,179.938,15.142,151.194
C04355=1105.268,304.014,-79.654,179.934,15.141,151.194
C04356=1105.262,303.767,-79.624,179.930,15.140,151.195
C04357=1105.254,303.388,-79.577,179.924,15.138,151.195
C04358=1105.245,303.008,-79.529,179.919,15.136,151.196
C04359=1105.236,302.629,-79.483,179.914,15.134,151.197
C04360=1105.228,302.250,-79.436,179.908,15.133,151.198
C04361=1105.223,302.002,-79.405,179.904,15.131,151.198
C04362=1105.217,301.754,-79.375,179.901,15.130,151.199
C04363=1105.210,301.505,-79.344,179.898,15.128,151.199
C04364=1105.205,301.257,-79.313,179.894,15.127,151.199
C04365=1105.200,301.009,-79.283,179.891,15.126,151.200
C04366=1105.194,300.762,-79.252,179.887,15.125,151.200
C04367=1105.189,300.513,-79.221,179.883,15.123,151.201
C04368=1105.183,300.266,-79.191,179.879,15.122,151.201
C04369=1105.177,300.017,-79.162,179.876,15.121,151.202
C04370=1105.172,299.769,-79.131,179.872,15.120,151.202
C04371=1105.166,299.521,-79.100,179.868,15.119,151.203
C04372=1105.161,299.273,-79.070,179.865,15.118,151.203
C04373=1105.156,299.025,-79.039,179.861,15.116,151.204
C04374=1105.150,298.777,-79.009,179.857,15.115,151.204
C04375=1105.144,298.529,-78.979,179.854,15.114,151.205
C04376=1105.138,298.281,-78.949,179.850,15.113,151.205
C04377=1105.133,298.033,-78.918,179.847,15.112,151.206
C04378=1105.128,297.785,-78.887,179.843,15.110,151.206
C04379=1105.122,297.537,-78.857,179.840,15.110,151.207
C04380=1105.116,297.289,-78.827,179.836,15.108,151.208
C04381=1105.110,297.041,-78.797,179.833,15.108,151.208
C04382=1105.105,296.793,-78.767,179.829,15.106,151.209
C04383=1105.098,296.545,-78.736,179.825,15.105,151.209
C04384=1105.093,296.296,-78.706,179.821,15.104,151.210
C04385=1105.088,296.048,-78.675,179.818,15.103,151.210
C04386=1105.082,295.800,-78.645,179.814,15.102,151.211
C04387=1105.076,295.552,-78.615,179.810,15.101,151.211
C04388=1105.070,295.304,-78.585,179.807,15.100,151.212
C04389=1105.065,295.056,-78.555,179.803,15.098,151.212
C04390=1105.059,294.808,-78.525,179.800,15.098,151.213
C04391=1105.053,294.560,-78.495,179.796,15.097,151.214
C04392=1105.048,294.312,-78.465,179.792,15.096,151.214
C04393=1105.042,294.064,-78.435,179.788,15.094,151.215
C04394=1105.036,293.815,-78.405,179.785,15.093,151.215
C04395=1105.031,293.568,-78.375,179.781,15.092,151.216
C04396=1105.025,293.319,-78.345,179.778,15.092,151.216
C04397=1105.019,293.071,-78.315,179.774,15.090,151.217
C04398=1105.014,292.823,-78.285,179.771,15.089,151.217
C04399=1105.008,292.575,-78.255,179.766,15.088,151.218
C04400=1105.003,292.327,-78.225,179.763,15.088,151.218
C04401=1104.997,292.079,-78.195,179.759,15.086,151.219
C04402=1104.992,291.831,-78.165,179.756,15.086,151.220
C04403=1104.985,291.583,-78.136,179.752,15.084,151.220
C04404=1104.980,291.335,-78.106,179.749,15.083,151.221
C04405=1104.974,291.087,-78.076,179.744,15.082,151.221
C04406=1104.968,290.839,-78.046,179.741,15.082,151.222
C04407=1104.963,290.590,-78.016,179.737,15.080,151.222
C04408=1104.957,290.343,-77.986,179.734,15.080,151.223
C04409=1104.949,289.977,-77.943,179.728,15.078,151.224
C04410=1104.941,289.612,-77.898,179.722,15.076,151.225
C04411=1104.932,289.246,-77.854,179.717,15.075,151.226
C04412=1104.923,288.880,-77.811,179.712,15.074,151.226
C04413=1104.918,288.632,-77.781,179.708,15.073,151.227
C04414=1104.911,288.384,-77.752,179.704,15.072,151.228
C04415=1104.906,288.137,-77.722,179.701,15.071,151.228
C04416=1104.901,287.888,-77.693,179.697,15.070,151.229
C04417=1104.895,287.640,-77.663,179.694,15.069,151.229
C04418=1104.889,287.392,-77.633,179.689,15.068,151.230
C04419=1104.883,287.144,-77.604,179.686,15.068,151.231
C04420=1104.878,286.895,-77.574,179.683,15.067,151.231
C04421=1104.872,286.647,-77.544,179.679,15.066,151.232
C04422=1104.866,286.399,-77.515,179.675,15.065,151.232
C04423=1104.861,286.151,-77.486,179.671,15.064,151.233
C04424=1104.856,285.903,-77.457,179.668,15.063,151.234
C04425=1104.849,285.655,-77.427,179.664,15.062,151.234
C04426=1104.844,285.407,-77.397,179.660,15.062,151.235
C04427=1104.838,285.158,-77.367,179.656,15.060,151.235
C04428=1104.833,284.910,-77.338,179.653,15.060,151.236
C04429=1104.827,284.662,-77.309,179.650,15.059,151.236
C04430=1104.821,284.414,-77.280,179.645,15.058,151.237
C04431=1104.816,284.165,-77.250,179.642,15.057,151.238
C04432=1104.810,283.917,-77.221,179.638,15.056,151.238
C04433=1104.804,283.669,-77.191,179.635,15.055,151.239
C04434=1104.799,283.421,-77.163,179.630,15.054,151.240
C04435=1104.793,283.173,-77.133,179.627,15.054,151.240
C04436=1104.787,282.925,-77.103,179.624,15.053,151.241
C04437=1104.781,282.676,-77.074,179.619,15.052,151.241
C04438=1104.776,282.429,-77.045,179.616,15.051,151.242
C04439=1104.771,282.180,-77.015,179.612,15.050,151.243
C04440=1104.765,281.932,-76.986,179.609,15.050,151.243
C04441=1104.759,281.683,-76.957,179.604,15.049,151.244
C04442=1104.754,281.436,-76.929,179.601,15.048,151.244
C04443=1104.748,281.187,-76.899,179.598,15.047,151.245
C04444=1104.742,280.939,-76.870,179.594,15.046,151.246
C04445=1104.736,280.691,-76.840,179.590,15.046,151.246
C04446=1104.731,280.443,-76.812,179.586,15.045,151.247
C04447=1104.726,280.194,-76.783,179.583,15.044,151.248
C04448=1104.719,279.946,-76.754,179.579,15.043,151.248
C04449=1104.714,279.698,-76.724,179.575,15.042,151.249
C04450=1104.708,279.450,-76.695,179.572,15.042,151.249
C04451=1104.703,279.202,-76.666,179.567,15.041,151.250
C04452=1104.697,278.953,-76.638,179.564,15.040,151.251
C04453=1104.691,278.704,-76.608,179.561,15.040,151.251
C04454=1104.686,278.457,-76.579,179.556,15.039,151.252
C04455=1104.680,278.208,-76.551,179.553,15.038,151.253
C04456=1104.674,277.960,-76.521,179.549,15.037,151.253
C04457=1104.668,277.712,-76.493,179.545,15.037,151.254
C04458=1104.663,277.463,-76.464,179.542,15.036,151.255
C04459=1104.657,277.215,-76.435,179.538,15.035,151.255
C04460=1104.651,276.968,-76.406,179.534,15.035,151.256
C04461=1104.643,276.611,-76.365,179.529,15.033,151.257
C04462=1104.635,276.255,-76.323,179.523,15.032,151.258
C04463=1104.627,275.899,-76.282,179.518,15.031,151.259
C04464=1104.619,275.543,-76.241,179.513,15.031,151.260
C04465=1104.613,275.295,-76.211,179.509,15.029,151.260
C04466=1104.608,275.047,-76.183,179.506,15.029,151.261
C04467=1104.602,274.798,-76.154,179.501,15.028,151.262
C04468=1104.596,274.550,-76.125,179.498,15.028,151.262
C04469=1104.591,274.302,-76.097,179.494,15.027,151.263
C04470=1104.585,274.054,-76.068,179.490,15.026,151.263
C04471=1104.579,273.806,-76.040,179.487,15.026,151.264
C04472=1104.574,273.557,-76.011,179.483,15.025,151.265
C04473=1104.568,273.309,-75.982,179.479,15.024,151.265
C04474=1104.563,273.060,-75.954,179.476,15.024,151.266
C04475=1104.556,272.812,-75.925,179.472,15.023,151.267
C04476=1104.551,272.563,-75.896,179.468,15.022,151.268
C04477=1104.546,272.315,-75.868,179.465,15.022,151.268
C04478=1104.540,272.067,-75.839,179.461,15.021,151.269
C04479=1104.534,271.819,-75.811,179.457,15.020,151.269
C04480=1104.528,271.571,-75.782,179.453,15.020,151.270
C04481=1104.523,271.323,-75.754,179.450,15.020,151.271
C04482=1104.517,271.074,-75.725,179.445,15.019,151.271
C04483=1104.511,270.826,-75.696,179.442,15.018,151.272
C04484=1104.506,270.578,-75.668,179.438,15.017,151.273
C04485=1104.500,270.329,-75.640,179.434,15.016,151.273
C04486=1104.494,270.081,-75.612,179.431,15.016,151.274
C04487=1104.488,269.833,-75.583,179.427,15.015,151.275
C04488=1104.483,269.585,-75.555,179.423,15.015,151.275
C04489=1104.477,269.336,-75.526,179.420,15.014,151.276
C04490=1104.472,269.088,-75.498,179.416,15.014,151.277
C04491=1104.466,268.839,-75.469,179.412,15.013,151.278
C04492=1104.460,268.591,-75.440,179.408,15.013,151.278
C04493=1104.455,268.343,-75.412,179.405,15.012,151.279
C04494=1104.449,268.094,-75.384,179.400,15.011,151.280
C04495=1104.444,267.846,-75.356,179.397,15.011,151.280
C04496=1104.438,267.597,-75.328,179.393,15.011,151.281
C04497=1104.432,267.349,-75.300,179.389,15.010,151.282
C04498=1104.426,267.100,-75.272,179.386,15.009,151.282
C04499=1104.421,266.853,-75.243,179.382,15.009,151.283
C04500=1104.415,266.604,-75.215,179.378,15.008,151.284
C04501=1104.409,266.356,-75.187,179.374,15.008,151.284
C04502=1104.403,266.107,-75.158,179.371,15.007,151.285
C04503=1104.398,265.859,-75.130,179.366,15.006,151.286
C04504=1104.392,265.610,-75.102,179.363,15.006,151.287
C04505=1104.387,265.362,-75.074,179.359,15.006,151.287
C04506=1104.381,265.114,-75.046,179.356,15.005,151.288
C04507=1104.376,264.866,-75.018,179.352,15.004,151.289
C04508=1104.370,264.618,-74.990,179.348,15.004,151.289
C04509=1104.364,264.369,-74.962,179.345,15.004,151.290
C04510=1104.358,264.121,-74.934,179.340,15.003,151.291
C04511=1104.352,263.872,-74.906,179.337,15.002,151.291
C04512=1104.347,263.624,-74.878,179.333,15.002,151.292
C04513=1104.339,263.271,-74.838,179.328,15.001,151.293
C04514=1104.330,262.917,-74.799,179.323,15.001,151.294
C04515=1104.322,262.565,-74.759,179.317,15.000,151.295
C04516=1104.314,262.211,-74.719,179.311,14.999,151.296
C04517=1104.308,261.963,-74.691,179.308,14.999,151.297
C04518=1104.302,261.714,-74.664,179.304,14.999,151.298
C04519=1104.297,261.466,-74.636,179.300,14.998,151.298
C04520=1104.291,261.218,-74.608,179.296,14.998,151.299
C04521=1104.285,260.969,-74.580,179.293,14.997,151.300
C04522=1104.279,260.721,-74.553,179.289,14.997,151.301
C04523=1104.274,260.472,-74.525,179.285,14.996,151.301
C04524=1104.268,260.224,-74.497,179.281,14.996,151.302
C04525=1104.262,259.976,-74.470,179.277,14.996,151.303
C04526=1104.256,259.727,-74.441,179.274,14.995,151.304
C04527=1104.251,259.479,-74.414,179.270,14.994,151.304
C04528=1104.245,259.230,-74.386,179.266,14.994,151.305
C04529=1104.239,258.982,-74.358,179.262,14.994,151.306
C04530=1104.234,258.734,-74.331,179.259,14.994,151.306
C04531=1104.227,258.485,-74.303,179.254,14.993,151.307
C04532=1104.222,258.237,-74.275,179.251,14.993,151.308
C04533=1104.217,257.988,-74.248,179.247,14.992,151.309
C04534=1104.210,257.740,-74.220,179.244,14.992,151.309
C04535=1104.205,257.491,-74.193,179.239,14.991,151.310
C04536=1104.200,257.243,-74.165,179.236,14.991,151.311
C04537=1104.193,256.995,-74.138,179.232,14.991,151.312
C04538=1104.188,256.746,-74.110,179.229,14.990,151.312
C04539=1104.183,256.498,-74.082,179.224,14.989,151.313
C04540=1104.177,256.249,-74.055,179.220,14.989,151.314
C04541=1104.171,256.001,-74.027,179.217,14.989,151.314
C04542=1104.165,255.753,-74.001,179.213,14.989,151.315
C04543=1104.159,255.504,-73.972,179.209,14.988,151.316
C04544=1104.154,255.256,-73.946,179.206,14.987,151.317
C04545=1104.148,255.007,-73.918,179.202,14.988,151.317
C04546=1104.143,254.759,-73.891,179.198,14.987,151.318
C04547=1104.137,254.510,-73.863,179.194,14.986,151.319
C04548=1104.132,254.262,-73.836,179.190,14.986,151.320
C04549=1104.126,254.013,-73.809,179.187,14.986,151.320
C04550=1104.120,253.765,-73.781,179.183,14.986,151.321
C04551=1104.114,253.516,-73.754,179.179,14.985,151.322
C04552=1104.109,253.268,-73.726,179.175,14.984,151.322
C04553=1104.103,253.020,-73.699,179.172,14.984,151.323
C04554=1104.098,252.771,-73.672,179.168,14.984,151.324
C04555=1104.092,252.523,-73.645,179.164,14.984,151.325
C04556=1104.086,252.274,-73.617,179.160,14.983,151.325
C04557=1104.080,252.026,-73.591,179.156,14.983,151.326
C04558=1104.075,251.777,-73.563,179.153,14.982,151.327
C04559=1104.069,251.529,-73.536,179.149,14.982,151.328
C04560=1104.064,251.281,-73.509,179.145,14.982,151.328
C04561=1104.058,251.032,-73.482,179.141,14.981,151.329
C04562=1104.053,250.783,-73.454,179.138,14.981,151.330
C04563=1104.047,250.535,-73.427,179.134,14.981,151.331
C04564=1104.042,250.286,-73.400,179.130,14.981,151.331
C04565=1104.034,249.931,-73.361,179.125,14.980,151.332
C04566=1104.025,249.575,-73.322,179.120,14.980,151.333
C04567=1104.018,249.219,-73.284,179.114,14.979,151.335
C04568=1104.009,248.862,-73.245,179.108,14.978,151.336
C04569=1104.004,248.614,-73.218,179.105,14.978,151.336
C04570=1103.998,248.366,-73.190,179.101,14.978,151.337
C04571=1103.993,248.117,-73.164,179.097,14.978,151.338
C04572=1103.988,247.869,-73.136,179.094,14.977,151.339
C04573=1103.982,247.620,-73.110,179.090,14.976,151.339
C04574=1103.976,247.372,-73.083,179.086,14.976,151.340
C04575=1103.971,247.123,-73.056,179.082,14.976,151.341
C04576=1103.965,246.875,-73.029,179.079,14.976,151.342
C04577=1103.959,246.626,-73.002,179.075,14.976,151.342
C04578=1103.953,246.377,-72.976,179.070,14.975,151.343
C04579=1103.948,246.129,-72.948,179.067,14.975,151.344
C04580=1103.942,245.880,-72.922,179.063,14.975,151.345
C04581=1103.936,245.632,-72.895,179.060,14.974,151.345
C04582=1103.931,245.384,-72.868,179.056,14.974,151.346
C04583=1103.926,245.135,-72.841,179.052,14.974,151.347
C04584=1103.920,244.887,-72.814,179.048,14.973,151.348
C04585=1103.914,244.638,-72.788,179.044,14.973,151.348
C04586=1103.908,244.390,-72.761,179.040,14.973,151.349
C04587=1103.904,244.141,-72.735,179.037,14.973,151.350
C04588=1103.898,243.892,-72.708,179.033,14.973,151.351
C04589=1103.892,243.644,-72.681,179.029,14.973,151.352
C04590=1103.886,243.396,-72.655,179.025,14.972,151.352
C04591=1103.880,243.147,-72.628,179.022,14.971,151.353
C04592=1103.874,242.898,-72.601,179.018,14.972,151.354
C04593=1103.868,242.650,-72.574,179.014,14.971,151.355
C04594=1103.864,242.400,-72.548,179.010,14.971,151.355
C04595=1103.858,242.152,-72.521,179.007,14.971,151.356
C04596=1103.852,241.904,-72.495,179.003,14.970,151.357
C04597=1103.846,241.655,-72.468,178.999,14.970,151.358
C04598=1103.841,241.406,-72.442,178.995,14.970,151.358
C04599=1103.835,241.158,-72.415,178.991,14.970,151.359
C04600=1103.829,240.910,-72.389,178.988,14.970,151.360
C04601=1103.823,240.661,-72.362,178.984,14.970,151.361
C04602=1103.818,240.412,-72.336,178.980,14.970,151.362
C04603=1103.812,240.164,-72.309,178.976,14.969,151.362
C04604=1103.806,239.916,-72.283,178.972,14.969,151.363
C04605=1103.801,239.667,-72.257,178.969,14.968,151.364
C04606=1103.795,239.418,-72.230,178.965,14.969,151.365
C04607=1103.789,239.170,-72.204,178.961,14.968,151.365
C04608=1103.784,238.921,-72.178,178.957,14.968,151.366
C04609=1103.778,238.673,-72.151,178.954,14.968,151.367
C04610=1103.772,238.424,-72.124,178.950,14.968,151.368
C04611=1103.767,238.175,-72.098,178.946,14.967,151.369
C04612=1103.761,237.927,-72.072,178.942,14.967,151.369
C04613=1103.756,237.678,-72.046,178.938,14.967,151.370
C04614=1103.750,237.430,-72.019,178.935,14.967,151.371
C04615=1103.744,237.181,-71.994,178.931,14.967,151.372
C04616=1103.738,236.933,-71.967,178.927,14.967,151.372
C04617=1103.730,236.569,-71.929,178.921,14.966,151.374
C04618=1103.722,236.207,-71.890,178.916,14.966,151.375
C04619=1103.714,235.845,-71.852,178.910,14.966,151.376
C04620=1103.706,235.482,-71.814,178.905,14.966,151.377
C04621=1103.700,235.233,-71.788,178.902,14.966,151.378
C04622=1103.694,234.984,-71.762,178.897,14.965,151.379
C04623=1103.689,234.736,-71.736,178.893,14.965,151.379
C04624=1103.684,234.488,-71.710,178.890,14.965,151.380
C04625=1103.677,234.239,-71.684,178.886,14.965,151.381
C04626=1103.672,233.991,-71.658,178.882,14.965,151.382
C04627=1103.666,233.742,-71.632,178.879,14.965,151.383
C04628=1103.661,233.493,-71.606,178.875,14.965,151.383
C04629=1103.655,233.245,-71.579,178.871,14.965,151.384
C04630=1103.649,232.996,-71.554,178.868,14.965,151.385
C04631=1103.644,232.748,-71.528,178.864,14.965,151.386
C04632=1103.638,232.499,-71.501,178.860,14.964,151.387
C04633=1103.633,232.250,-71.476,178.856,14.964,151.387
C04634=1103.626,232.002,-71.450,178.852,14.964,151.388
C04635=1103.621,231.753,-71.424,178.848,14.964,151.389
C04636=1103.615,231.504,-71.398,178.845,14.963,151.390
C04637=1103.610,231.256,-71.372,178.841,14.964,151.391
C04638=1103.604,231.007,-71.347,178.837,14.963,151.391
C04639=1103.599,230.758,-71.321,178.833,14.963,151.392
C04640=1103.593,230.510,-71.294,178.830,14.963,151.393
C04641=1103.587,230.261,-71.269,178.826,14.963,151.394
C04642=1103.581,230.012,-71.243,178.822,14.963,151.394
C04643=1103.576,229.764,-71.217,178.819,14.963,151.395
C04644=1103.570,229.515,-71.192,178.814,14.962,151.396
C04645=1103.565,229.266,-71.166,178.810,14.962,151.397
C04646=1103.558,229.018,-71.140,178.807,14.963,151.398
C04647=1103.553,228.769,-71.114,178.803,14.962,151.399
C04648=1103.548,228.521,-71.088,178.799,14.962,151.399
C04649=1103.542,228.272,-71.063,178.796,14.962,151.400
C04650=1103.536,228.023,-71.037,178.792,14.962,151.401
C04651=1103.530,227.775,-71.012,178.788,14.962,151.402
C04652=1103.524,227.526,-70.986,178.784,14.962,151.403
C04653=1103.519,227.278,-70.961,178.780,14.962,151.403
C04654=1103.513,227.029,-70.935,178.777,14.962,151.404
C04655=1103.507,226.780,-70.910,178.773,14.962,151.405
C04656=1103.502,226.531,-70.884,178.769,14.962,151.406
C04657=1103.497,226.283,-70.858,178.766,14.962,151.407
C04658=1103.491,226.034,-70.833,178.762,14.962,151.407
C04659=1103.485,225.785,-70.807,178.758,14.962,151.408
C04660=1103.480,225.537,-70.782,178.754,14.962,151.409
C04661=1103.474,225.288,-70.756,178.750,14.961,151.410
C04662=1103.468,225.040,-70.731,178.746,14.961,151.411
C04663=1103.462,224.791,-70.705,178.743,14.961,151.411
C04664=1103.457,224.543,-70.680,178.739,14.961,151.412
C04665=1103.451,224.294,-70.654,178.735,14.961,151.413
C04666=1103.445,224.045,-70.629,178.731,14.961,151.414
C04667=1103.440,223.796,-70.604,178.727,14.961,151.415
C04668=1103.434,223.547,-70.578,178.724,14.961,151.416
C04669=1103.426,223.177,-70.541,178.719,14.962,151.417
C04670=1103.418,222.806,-70.502,178.713,14.961,151.418
C04671=1103.409,222.435,-70.465,178.707,14.962,151.419
C04672=1103.401,222.063,-70.427,178.702,14.961,151.420
C04673=1103.395,221.814,-70.402,178.698,14.961,151.421
C04674=1103.390,221.566,-70.376,178.694,14.961,151.422
C04675=1103.384,221.317,-70.351,178.690,14.961,151.423
C04676=1103.378,221.068,-70.326,178.686,14.961,151.424
C04677=1103.372,220.820,-70.301,178.683,14.961,151.425
C04678=1103.367,220.571,-70.275,178.679,14.961,151.425
C04679=1103.361,220.322,-70.251,178.675,14.961,151.426
C04680=1103.355,220.074,-70.226,178.672,14.961,151.427
C04681=1103.350,219.825,-70.200,178.668,14.961,151.428
C04682=1103.344,219.576,-70.174,178.664,14.961,151.429
C04683=1103.338,219.328,-70.150,178.660,14.961,151.429
C04684=1103.332,219.079,-70.125,178.656,14.961,151.430
C04685=1103.328,218.830,-70.100,178.653,14.961,151.431
C04686=1103.321,218.581,-70.075,178.649,14.961,151.432
C04687=1103.315,218.333,-70.049,178.645,14.961,151.433
C04688=1103.310,218.084,-70.025,178.641,14.962,151.434
C04689=1103.304,217.835,-70.000,178.638,14.961,151.434
C04690=1103.299,217.587,-69.975,178.634,14.961,151.435
C04691=1103.293,217.338,-69.950,178.630,14.961,151.436
C04692=1103.287,217.090,-69.925,178.626,14.961,151.437
C04693=1103.281,216.841,-69.900,178.623,14.962,151.438
C04694=1103.276,216.593,-69.875,178.619,14.961,151.438
C04695=1103.271,216.343,-69.850,178.615,14.962,151.439
C04696=1103.264,216.094,-69.824,178.611,14.962,151.440
C04697=1103.259,215.846,-69.800,178.608,14.961,151.441
C04698=1103.253,215.597,-69.775,178.604,14.962,151.442
C04699=1103.248,215.349,-69.751,178.600,14.961,151.443
C04700=1103.242,215.099,-69.725,178.596,14.962,151.443
C04701=1103.237,214.851,-69.700,178.593,14.962,151.444
C04702=1103.231,214.602,-69.676,178.589,14.962,151.445
C04703=1103.225,214.354,-69.651,178.585,14.962,151.446
C04704=1103.219,214.104,-69.626,178.582,14.961,151.447
C04705=1103.214,213.856,-69.602,178.578,14.962,151.447
C04706=1103.209,213.608,-69.577,178.574,14.962,151.448
C04707=1103.203,213.359,-69.552,178.570,14.962,151.449
C04708=1103.197,213.111,-69.527,178.566,14.962,151.450
C04709=1103.191,212.861,-69.503,178.563,14.962,151.451
C04710=1103.187,212.612,-69.478,178.559,14.962,151.452
C04711=1103.180,212.364,-69.453,178.555,14.962,151.452
C04712=1103.175,212.115,-69.428,178.551,14.962,151.453
C04713=1103.169,211.866,-69.404,178.548,14.962,151.454
C04714=1103.164,211.617,-69.379,178.544,14.962,151.455
C04715=1103.158,211.369,-69.354,178.540,14.962,151.456
C04716=1103.152,211.120,-69.330,178.536,14.962,151.457
C04717=1103.146,210.871,-69.305,178.533,14.962,151.457
C04718=1103.140,210.623,-69.282,178.529,14.962,151.458
C04719=1103.135,210.375,-69.257,178.525,14.962,151.459
C04720=1103.129,210.125,-69.232,178.521,14.962,151.460
C04721=1103.121,209.758,-69.195,178.516,14.963,151.461
C04722=1103.112,209.390,-69.159,178.511,14.963,151.462
C04723=1103.104,209.022,-69.123,178.505,14.963,151.464
C04724=1103.096,208.655,-69.087,178.499,14.963,151.465
C04725=1103.073,207.654,-68.990,178.468,14.958,151.471
C04726=1103.067,207.405,-68.965,178.464,14.959,151.472
C04727=1103.062,207.156,-68.941,178.460,14.960,151.473
C04728=1103.056,206.908,-68.917,178.456,14.961,151.474
C04729=1103.050,206.659,-68.893,178.452,14.962,151.475
C04730=1103.045,206.410,-68.868,178.448,14.963,151.476
C04731=1103.039,206.162,-68.844,178.444,14.964,151.477
C04732=1103.033,205.913,-68.820,178.440,14.965,151.478
C04733=1103.027,205.664,-68.796,178.436,14.965,151.479
C04734=1103.022,205.416,-68.771,178.432,14.967,151.480
C04735=1103.016,205.166,-68.747,178.428,14.967,151.481
C04736=1103.010,204.918,-68.723,178.424,14.968,151.482
C04737=1103.005,204.669,-68.699,178.421,14.969,151.483
C04738=1102.999,204.420,-68.674,178.416,14.970,151.484
C04739=1102.993,204.171,-68.651,178.412,14.971,151.486
C04740=1102.988,203.923,-68.627,178.408,14.972,151.487
C04741=1102.983,203.674,-68.603,178.404,14.973,151.488
C04742=1102.976,203.425,-68.579,178.400,14.973,151.489
C04743=1102.971,203.176,-68.555,178.396,14.975,151.490
C04744=1102.965,202.928,-68.530,178.392,14.975,151.491
C04745=1102.959,202.678,-68.507,178.388,14.976,151.492
C04746=1102.954,202.430,-68.483,178.385,14.977,151.493
C04747=1102.948,202.181,-68.459,178.380,14.978,151.494
C04748=1102.942,201.933,-68.435,178.376,14.979,151.495
C04749=1102.936,201.684,-68.411,178.373,14.980,151.496
C04750=1102.931,201.435,-68.387,178.369,14.981,151.497
C04751=1102.925,201.186,-68.364,178.364,14.981,151.498
C04752=1102.919,200.937,-68.339,178.361,14.983,151.499
C04753=1102.913,200.688,-68.316,178.357,14.983,151.500
C04754=1102.908,200.440,-68.292,178.353,14.985,151.502
C04755=1102.902,200.191,-68.268,178.349,14.986,151.503
C04756=1102.896,199.942,-68.243,178.345,14.986,151.504
C04757=1102.890,199.693,-68.221,178.341,14.988,151.505
C04758=1102.885,199.445,-68.196,178.337,14.988,151.506
C04759=1102.879,199.196,-68.173,178.333,14.989,151.507
C04760=1102.873,198.946,-68.149,178.329,14.990,151.508
C04761=1102.867,198.698,-68.125,178.325,14.991,151.509
C04762=1102.862,198.449,-68.102,178.321,14.991,151.510
C04763=1102.856,198.201,-68.078,178.317,14.993,151.511
C04764=1102.850,197.952,-68.054,178.313,14.993,151.512
C04765=1102.845,197.702,-68.030,178.309,14.994,151.513
C04766=1102.838,197.454,-68.007,178.306,14.995,151.514
C04767=1102.833,197.205,-67.983,178.302,14.996,151.515
C04768=1102.827,196.957,-67.959,178.298,14.996,151.516
C04769=1102.822,196.708,-67.936,178.294,14.998,151.517
C04770=1102.816,196.458,-67.912,178.290,14.998,151.518
C04771=1102.810,196.210,-67.889,178.286,14.999,151.519
C04772=1102.805,195.961,-67.865,178.282,15.000,151.520
C04773=1102.799,195.712,-67.842,178.278,15.001,151.521
C04774=1102.793,195.464,-67.818,178.274,15.002,151.523
C04775=1102.788,195.215,-67.795,178.270,15.003,151.524
C04776=1102.781,194.966,-67.770,178.266,15.003,151.524
C04777=1102.776,194.717,-67.748,178.263,15.004,151.526
C04778=1102.770,194.468,-67.723,178.259,15.005,151.527
C04779=1102.765,194.219,-67.700,178.255,15.006,151.528
C04780=1102.759,193.970,-67.677,178.251,15.007,151.529
C04781=1102.754,193.722,-67.653,178.247,15.008,151.530
C04782=1102.748,193.473,-67.630,178.243,15.008,151.531
C04783=1102.742,193.225,-67.607,178.240,15.009,151.532
C04784=1102.737,192.975,-67.583,178.235,15.010,151.533
C04785=1102.731,192.726,-67.560,178.231,15.011,151.534
C04786=1102.725,192.454,-67.534,178.227,15.011,151.535
C04787=1102.718,192.182,-67.509,178.223,15.013,151.536
C04788=1102.712,191.910,-67.482,178.219,15.014,151.537
C04789=1102.706,191.638,-67.458,178.215,15.015,151.538
C04790=1102.700,191.389,-67.435,178.211,15.015,151.539
C04791=1102.695,191.141,-67.411,178.206,15.016,151.540
C04792=1102.689,190.892,-67.388,178.203,15.017,151.541
C04793=1102.684,190.643,-67.365,178.199,15.017,151.542
C04794=1102.679,190.394,-67.341,178.196,15.019,151.543
C04795=1102.673,190.145,-67.317,178.192,15.019,151.544
C04796=1102.667,189.897,-67.295,178.188,15.020,151.545
C04797=1102.661,189.648,-67.272,178.184,15.021,151.546
C04798=1102.656,189.398,-67.248,178.180,15.021,151.547
C04799=1102.650,189.150,-67.225,178.176,15.022,151.548
C04800=1102.645,188.901,-67.202,178.173,15.023,151.549
C04801=1102.639,188.652,-67.178,178.169,15.024,151.550
C04802=1102.633,188.403,-67.156,178.165,15.024,151.551
C04803=1102.628,188.154,-67.132,178.161,15.026,151.552
C04804=1102.622,187.905,-67.109,178.157,15.026,151.553
C04805=1102.617,187.656,-67.086,178.153,15.027,151.554
C04806=1102.611,187.408,-67.063,178.150,15.028,151.555
C04807=1102.605,187.159,-67.040,178.146,15.028,151.556
C04808=1102.600,186.909,-67.017,178.142,15.029,151.557
C04809=1102.594,186.661,-66.994,178.138,15.030,151.558
C04810=1102.589,186.412,-66.971,178.134,15.030,151.559
C04811=1102.583,186.163,-66.948,178.131,15.031,151.560
C04812=1102.577,185.914,-66.925,178.127,15.032,151.561
C04813=1102.571,185.665,-66.902,178.123,15.032,151.562
C04814=1102.567,185.416,-66.879,178.120,15.034,151.563
C04815=1102.561,185.168,-66.856,178.115,15.034,151.564
C04816=1102.556,184.919,-66.833,178.111,15.035,151.565
C04817=1102.550,184.670,-66.810,178.108,15.036,151.566
C04818=1102.543,184.421,-66.788,178.104,15.037,151.567
C04819=1102.538,184.172,-66.765,178.101,15.038,151.568
C04820=1102.532,183.923,-66.742,178.096,15.038,151.569
C04821=1102.526,183.675,-66.719,178.092,15.039,151.570
C04822=1102.520,183.426,-66.696,178.089,15.040,151.571
C04823=1102.515,183.177,-66.673,178.085,15.041,151.572
C04824=1102.509,182.928,-66.650,178.081,15.041,151.573
C04825=1102.503,182.679,-66.627,178.078,15.042,151.574
C04826=1102.497,182.430,-66.605,178.073,15.043,151.575
C04827=1102.491,182.181,-66.582,178.070,15.044,151.576
C04828=1102.485,181.933,-66.559,178.066,15.044,151.577
C04829=1102.480,181.683,-66.536,178.062,15.045,151.578
C04830=1102.474,181.434,-66.514,178.059,15.046,151.579
C04831=1102.468,181.185,-66.491,178.055,15.047,151.580
C04832=1102.462,180.937,-66.468,178.051,15.048,151.581
C04833=1102.456,180.688,-66.445,178.047,15.048,151.582
C04834=1102.451,180.438,-66.423,178.043,15.049,151.583
C04835=1102.445,180.189,-66.400,178.040,15.050,151.584
C04836=1102.439,179.940,-66.377,178.036,15.051,151.585
C04837=1102.433,179.693,-66.355,178.032,15.051,151.586
C04838=1102.428,179.444,-66.332,178.028,15.052,151.587
C04839=1102.422,179.194,-66.310,178.024,15.053,151.588
C04840=1102.417,178.945,-66.287,178.021,15.054,151.589
C04841=1102.411,178.696,-66.264,178.017,15.054,151.590
C04842=1102.405,178.447,-66.242,178.013,15.055,151.591
C04843=1102.399,178.198,-66.220,178.010,15.056,151.592
C04844=1102.393,177.949,-66.197,178.006,15.057,151.593
C04845=1102.388,177.701,-66.175,178.002,15.058,151.594
C04846=1102.382,177.452,-66.152,177.998,15.058,151.595
C04847=1102.376,177.203,-66.129,177.994,15.059,151.596
C04848=1102.371,176.954,-66.107,177.991,15.059,151.597
C04849=1102.365,176.705,-66.084,177.987,15.060,151.598
C04850=1102.359,176.433,-66.060,177.983,15.061,151.599
C04851=1102.353,176.160,-66.035,177.979,15.062,151.600
C04852=1102.346,175.888,-66.010,177.976,15.063,151.601
C04853=1102.340,175.615,-65.986,177.971,15.063,151.602
C04854=1102.334,175.367,-65.964,177.967,15.064,151.603
C04855=1102.329,175.117,-65.942,177.963,15.064,151.604
C04856=1102.323,174.869,-65.919,177.960,15.065,151.605
C04857=1102.317,174.620,-65.898,177.956,15.066,151.606
C04858=1102.312,174.371,-65.875,177.953,15.067,151.607
C04859=1102.306,174.121,-65.852,177.949,15.067,151.608
C04860=1102.300,173.873,-65.830,177.945,15.068,151.609
C04861=1102.295,173.624,-65.808,177.942,15.069,151.609
C04862=1102.289,173.375,-65.785,177.938,15.069,151.610
C04863=1102.283,173.126,-65.764,177.934,15.070,151.611
C04864=1102.278,172.878,-65.741,177.930,15.071,151.612
C04865=1102.272,172.628,-65.719,177.926,15.071,151.613
C04866=1102.266,172.379,-65.697,177.923,15.072,151.614
C04867=1102.260,172.130,-65.674,177.919,15.073,151.615
C04868=1102.256,171.881,-65.652,177.916,15.074,151.616
C04869=1102.249,171.633,-65.630,177.912,15.074,151.617
C04870=1102.244,171.383,-65.608,177.908,15.074,151.618
C04871=1102.238,171.135,-65.587,177.905,15.076,151.619
C04872=1102.232,170.886,-65.564,177.901,15.076,151.620
C04873=1102.227,170.636,-65.541,177.898,15.077,151.621
C04874=1102.221,170.388,-65.520,177.894,15.077,151.622
C04875=1102.216,170.139,-65.497,177.890,15.077,151.622
C04876=1102.210,169.890,-65.475,177.887,15.078,151.623
C04877=1102.205,169.641,-65.454,177.883,15.079,151.624
C04878=1102.199,169.392,-65.431,177.879,15.079,151.625
C04879=1102.193,169.143,-65.409,177.876,15.080,151.626
C04880=1102.188,168.894,-65.387,177.872,15.081,151.627
C04881=1102.182,168.645,-65.366,177.869,15.082,151.628
C04882=1102.176,168.396,-65.343,177.865,15.082,151.629
C04883=1102.171,168.147,-65.321,177.861,15.082,151.630
C04884=1102.165,167.898,-65.299,177.858,15.083,151.631
C04885=1102.160,167.649,-65.278,177.854,15.083,151.632
C04886=1102.154,167.400,-65.256,177.851,15.084,151.633
C04887=1102.148,167.151,-65.233,177.847,15.085,151.634
C04888=1102.143,166.902,-65.211,177.843,15.085,151.634
C04889=1102.137,166.653,-65.189,177.839,15.086,151.635
C04890=1102.132,166.404,-65.168,177.836,15.087,151.636
C04891=1102.126,166.155,-65.146,177.832,15.088,151.637
C04892=1102.121,165.906,-65.124,177.829,15.088,151.638
C04893=1102.115,165.657,-65.102,177.825,15.088,151.639
C04894=1102.109,165.408,-65.080,177.822,15.089,151.640
C04895=1102.104,165.159,-65.058,177.818,15.089,151.641
C04896=1102.098,164.910,-65.036,177.815,15.090,151.642
C04897=1102.093,164.661,-65.014,177.811,15.091,151.643
C04898=1102.087,164.412,-64.993,177.807,15.091,151.643
C04899=1102.082,164.163,-64.971,177.804,15.091,151.644
C04900=1102.076,163.914,-64.949,177.800,15.092,151.645
C04901=1102.070,163.666,-64.928,177.797,15.093,151.646
C04902=1102.065,163.416,-64.906,177.793,15.093,151.647
C04903=1102.060,163.168,-64.885,177.789,15.093,151.648
C04904=1102.054,162.918,-64.862,177.786,15.094,151.649
C04905=1102.049,162.670,-64.841,177.782,15.095,151.650
C04906=1102.043,162.420,-64.819,177.779,15.096,151.650
C04907=1102.038,162.172,-64.798,177.775,15.096,151.651
C04908=1102.032,161.922,-64.775,177.772,15.096,151.652
C04909=1102.027,161.674,-64.754,177.768,15.097,151.653
C04910=1102.020,161.424,-64.732,177.765,15.097,151.654
C04911=1102.015,161.176,-64.711,177.761,15.098,151.655
C04912=1102.009,160.926,-64.689,177.758,15.098,151.656
C04913=1102.004,160.677,-64.668,177.754,15.099,151.657
C04914=1101.997,160.404,-64.645,177.750,15.100,151.658
C04915=1101.991,160.132,-64.621,177.746,15.100,151.659
C04916=1101.985,159.859,-64.597,177.742,15.101,151.659
C04917=1101.979,159.587,-64.574,177.738,15.101,151.661
C04918=1101.973,159.337,-64.552,177.734,15.102,151.661
C04919=1101.967,159.089,-64.531,177.732,15.102,151.662
C04920=1101.962,158.839,-64.509,177.728,15.103,151.663
C04921=1101.957,158.590,-64.488,177.725,15.104,151.664
C04922=1101.950,158.341,-64.467,177.721,15.104,151.665
C04923=1101.945,158.092,-64.445,177.718,15.105,151.666
C04924=1101.939,157.843,-64.424,177.714,15.105,151.667
C04925=1101.934,157.594,-64.402,177.710,15.105,151.668
C04926=1101.928,157.345,-64.381,177.707,15.106,151.668
C04927=1101.922,157.096,-64.360,177.703,15.106,151.669
C04928=1101.916,156.847,-64.338,177.700,15.107,151.670
C04929=1101.911,156.598,-64.317,177.696,15.108,151.671
C04930=1101.905,156.349,-64.296,177.693,15.109,151.672
C04931=1101.899,156.100,-64.274,177.689,15.108,151.673
C04932=1101.894,155.851,-64.253,177.685,15.109,151.674
C04933=1101.889,155.601,-64.232,177.682,15.110,151.674
C04934=1101.883,155.353,-64.210,177.678,15.110,151.675
C04935=1101.877,155.104,-64.189,177.676,15.111,151.676
C04936=1101.872,154.855,-64.168,177.672,15.111,151.677
C04937=1101.865,154.605,-64.147,177.668,15.111,151.678
C04938=1101.860,154.357,-64.125,177.665,15.112,151.679
C04939=1101.855,154.108,-64.105,177.661,15.113,151.680
C04940=1101.849,153.859,-64.083,177.658,15.113,151.680
C04941=1101.843,153.609,-64.063,177.654,15.113,151.681
C04942=1101.837,153.360,-64.041,177.651,15.114,151.682
C04943=1101.832,153.112,-64.020,177.647,15.114,151.683
C04944=1101.826,152.863,-63.999,177.644,15.115,151.684
C04945=1101.820,152.613,-63.977,177.640,15.116,151.685
C04946=1101.815,152.364,-63.957,177.637,15.115,151.685
C04947=1101.809,152.116,-63.936,177.634,15.116,151.686
C04948=1101.803,151.866,-63.915,177.630,15.117,151.687
C04949=1101.798,151.617,-63.893,177.627,15.117,151.688
C04950=1101.792,151.368,-63.873,177.623,15.118,151.689
C04951=1101.786,151.119,-63.851,177.619,15.118,151.690
C04952=1101.781,150.870,-63.831,177.616,15.118,151.691
C04953=1101.775,150.621,-63.809,177.613,15.119,151.691
C04954=1101.770,150.372,-63.789,177.610,15.119,151.692
C04955=1101.764,150.123,-63.767,177.606,15.120,151.693
C04956=1101.758,149.873,-63.746,177.603,15.121,151.694
C04957=1101.753,149.625,-63.725,177.599,15.121,151.695
C04958=1101.748,149.376,-63.705,177.595,15.121,151.696
C04959=1101.741,149.126,-63.684,177.592,15.121,151.696
C04960=1101.735,148.878,-63.663,177.589,15.122,151.697
C04961=1101.730,148.629,-63.642,177.585,15.123,151.698
C04962=1101.725,148.380,-63.621,177.582,15.123,151.699
C04963=1101.719,148.130,-63.600,177.579,15.124,151.700
C04964=1101.713,147.881,-63.580,177.575,15.123,151.701
C04965=1101.708,147.633,-63.558,177.571,15.124,151.701
C04966=1101.701,147.383,-63.538,177.568,15.124,151.702
C04967=1101.696,147.134,-63.517,177.565,15.125,151.703
C04968=1101.690,146.885,-63.496,177.562,15.125,151.704
C04969=1101.685,146.636,-63.475,177.558,15.126,151.705
C04970=1101.679,146.387,-63.455,177.555,15.126,151.705
C04971=1101.673,146.138,-63.434,177.551,15.126,151.706
C04972=1101.667,145.888,-63.413,177.548,15.127,151.707
C04973=1101.662,145.639,-63.393,177.544,15.127,151.708
C04974=1101.657,145.390,-63.372,177.541,15.127,151.709
C04975=1101.650,145.142,-63.351,177.538,15.128,151.710
C04976=1101.645,144.892,-63.330,177.534,15.128,151.710
C04977=1101.639,144.643,-63.310,177.531,15.129,151.711
C04978=1101.633,144.370,-63.287,177.527,15.129,151.712
C04979=1101.626,144.097,-63.264,177.523,15.130,151.713
C04980=1101.621,143.824,-63.242,177.520,15.130,151.714
C04981=1101.614,143.551,-63.220,177.517,15.131,151.715
C04982=1101.609,143.302,-63.199,177.513,15.131,151.716
C04983=1101.603,143.052,-63.178,177.509,15.131,151.716
C04984=1101.597,142.804,-63.158,177.506,15.131,151.717
C04985=1101.592,142.555,-63.137,177.502,15.132,151.718
C04986=1101.587,142.306,-63.117,177.500,15.132,151.719
C04987=1101.581,142.057,-63.097,177.496,15.133,151.720
C04988=1101.575,141.807,-63.076,177.493,15.133,151.720
C04989=1101.569,141.558,-63.055,177.489,15.133,151.721
C04990=1101.563,141.309,-63.035,177.487,15.134,151.722
C04991=1101.558,141.060,-63.015,177.483,15.134,151.723
C04992=1101.553,140.811,-62.994,177.479,15.134,151.723
C04993=1101.547,140.562,-62.974,177.476,15.135,151.724
C04994=1101.541,140.312,-62.953,177.472,15.135,151.725
C04995=1101.536,140.063,-62.933,177.470,15.135,151.726
C04996=1101.530,139.814,-62.913,177.466,15.135,151.727
C04997=1101.524,139.566,-62.891,177.463,15.136,151.727
C04998=1101.518,139.317,-62.871,177.459,15.136,151.728
C04999=1101.512,139.067,-62.850,177.456,15.137,151.729
C05000=1101.507,138.818,-62.831,177.453,15.137,151.730
C05001=1101.502,138.569,-62.811,177.449,15.137,151.731
C05002=1101.496,138.320,-62.790,177.446,15.138,151.731
C05003=1101.490,138.071,-62.770,177.443,15.138,151.732
C05004=1101.485,137.822,-62.750,177.439,15.139,151.733
C05005=1101.479,137.573,-62.730,177.436,15.138,151.734
C05006=1101.473,137.323,-62.709,177.433,15.139,151.734
C05007=1101.467,137.074,-62.689,177.430,15.139,151.735
C05008=1101.462,136.825,-62.668,177.426,15.140,151.736
C05009=1101.456,136.576,-62.648,177.423,15.140,151.737
C05010=1101.451,136.327,-62.628,177.420,15.140,151.738
C05011=1101.445,136.078,-62.608,177.416,15.140,151.738
C05012=1101.440,135.829,-62.588,177.413,15.140,151.739
C05013=1101.434,135.580,-62.568,177.410,15.141,151.740
C05014=1101.428,135.331,-62.548,177.406,15.141,151.741
C05015=1101.422,135.081,-62.527,177.403,15.142,151.741
C05016=1101.416,134.832,-62.507,177.400,15.142,151.742
C05017=1101.411,134.583,-62.487,177.397,15.142,151.743
C05018=1101.405,134.334,-62.467,177.393,15.142,151.744
C05019=1101.400,134.085,-62.447,177.391,15.143,151.744
C05020=1101.394,133.836,-62.427,177.387,15.143,151.745
C05021=1101.388,133.587,-62.406,177.384,15.144,151.746
C05022=1101.382,133.338,-62.386,177.380,15.143,151.747
C05023=1101.377,133.089,-62.367,177.377,15.144,151.748
C05024=1101.371,132.839,-62.346,177.374,15.144,151.748
C05025=1101.365,132.591,-62.327,177.370,15.144,151.749
C05026=1101.361,132.341,-62.307,177.368,15.144,151.750
C05027=1101.355,132.092,-62.287,177.364,15.144,151.750
C05028=1101.349,131.843,-62.267,177.361,15.145,151.751
C05029=1101.343,131.594,-62.246,177.358,15.145,151.752
C05030=1101.338,131.345,-62.227,177.355,15.145,151.753
C05031=1101.332,131.096,-62.207,177.351,15.145,151.753
C05032=1101.325,130.846,-62.187,177.348,15.146,151.754
C05033=1101.320,130.597,-62.167,177.344,15.146,151.755
C05034=1101.314,130.348,-62.147,177.342,15.147,151.756
C05035=1101.308,130.098,-62.128,177.338,15.147,151.757
C05036=1101.302,129.850,-62.108,177.335,15.147,151.757
C05037=1101.296,129.601,-62.088,177.332,15.147,151.758
C05038=1101.291,129.351,-62.068,177.329,15.148,151.759
C05039=1101.285,129.102,-62.048,177.325,15.148,151.760
C05040=1101.279,128.853,-62.028,177.322,15.148,151.760
C05041=1101.274,128.604,-62.009,177.319,15.148,151.761
C05042=1101.268,128.331,-61.987,177.315,15.148,151.762
C05043=1101.261,128.058,-61.966,177.311,15.148,151.763
C05044=1101.256,127.784,-61.944,177.309,15.149,151.763
C05045=1101.249,127.512,-61.922,177.305,15.149,151.764
C05046=1101.243,127.263,-61.902,177.301,15.149,151.765
C05047=1101.238,127.013,-61.883,177.299,15.149,151.766
C05048=1101.232,126.764,-61.863,177.295,15.149,151.766
C05049=1101.226,126.515,-61.843,177.292,15.150,151.767
C05050=1101.220,126.266,-61.823,177.289,15.150,151.768
C05051=1101.215,126.017,-61.804,177.286,15.150,151.769
C05052=1101.209,125.767,-61.785,177.282,15.150,151.769
C05053=1101.203,125.518,-61.765,177.279,15.151,151.770
C05054=1101.198,125.269,-61.745,177.276,15.151,151.771
C05055=1101.192,125.020,-61.725,177.273,15.151,151.771
C05056=1101.186,124.770,-61.706,177.270,15.151,151.772
C05057=1101.180,124.521,-61.686,177.267,15.151,151.773
C05058=1101.175,124.272,-61.667,177.263,15.151,151.774
C05059=1101.169,124.023,-61.647,177.261,15.152,151.774
C05060=1101.163,123.774,-61.627,177.257,15.152,151.775
C05061=1101.158,123.525,-61.609,177.255,15.152,151.776
C05062=1101.153,123.275,-61.589,177.251,15.152,151.776
C05063=1101.147,123.026,-61.569,177.248,15.153,151.777
C05064=1101.141,122.777,-61.550,177.245,15.152,151.778
C05065=1101.136,122.528,-61.530,177.241,15.152,151.779
C05066=1101.130,122.279,-61.510,177.238,15.153,151.779
C05067=1101.124,122.029,-61.491,177.235,15.152,151.780
C05068=1101.118,121.780,-61.472,177.232,15.153,151.781
C05069=1101.113,121.532,-61.452,177.229,15.153,151.781
C05070=1101.107,121.282,-61.433,177.226,15.153,151.782
C05071=1101.101,121.033,-61.414,177.222,15.153,151.783
C05072=1101.096,120.784,-61.395,177.220,15.154,151.784
C05073=1101.090,120.535,-61.375,177.216,15.153,151.784
C05074=1101.084,120.285,-61.355,177.214,15.154,151.785
C05075=1101.079,120.037,-61.336,177.210,15.154,151.786
C05076=1101.073,119.787,-61.317,177.207,15.154,151.786
C05077=1101.068,119.538,-61.298,177.204,15.154,151.787
C05078=1101.062,119.289,-61.278,177.201,15.154,151.788
C05079=1101.056,119.039,-61.259,177.198,15.154,151.788
C05080=1101.051,118.791,-61.240,177.195,15.154,151.789
C05081=1101.045,118.541,-61.221,177.191,15.154,151.790
C05082=1101.040,118.292,-61.201,177.189,15.154,151.790
C05083=1101.034,118.042,-61.182,177.185,15.154,151.791
C05084=1101.028,117.793,-61.163,177.183,15.154,151.792
C05085=1101.023,117.545,-61.143,177.179,15.154,151.792
C05086=1101.017,117.295,-61.124,177.176,15.155,151.793
C05087=1101.011,117.046,-61.105,177.173,15.154,151.794
C05088=1101.006,116.797,-61.086,177.170,15.155,151.794
C05089=1101.001,116.548,-61.067,177.167,15.154,151.795
C05090=1100.995,116.298,-61.047,177.164,15.155,151.796
C05091=1100.989,116.049,-61.028,177.161,15.155,151.796
C05092=1100.984,115.800,-61.009,177.158,15.155,151.797
C05093=1100.978,115.551,-60.990,177.155,15.155,151.798
C05094=1100.973,115.301,-60.971,177.152,15.155,151.798
C05095=1100.967,115.052,-60.952,177.149,15.155,151.799
C05096=1100.962,114.803,-60.933,177.145,15.155,151.800
C05097=1100.956,114.554,-60.914,177.143,15.155,151.800
C05098=1100.951,114.304,-60.894,177.139,15.155,151.801
C05099=1100.945,114.055,-60.875,177.137,15.155,151.802
C05100=1100.939,113.807,-60.857,177.133,15.155,151.802
C05101=1100.933,113.557,-60.838,177.131,15.155,151.803
C05102=1100.928,113.308,-60.818,177.127,15.155,151.804
C05103=1100.922,113.058,-60.799,177.125,15.155,151.804
C05104=1100.917,112.809,-60.780,177.121,15.155,151.805
C05105=1100.911,112.560,-60.761,177.119,15.155,151.806
C05106=1100.904,112.287,-60.741,177.115,15.155,151.806
C05107=1100.898,112.013,-60.720,177.112,15.156,151.807
C05108=1100.892,111.741,-60.699,177.109,15.156,151.808
C05109=1100.886,111.467,-60.679,177.105,15.155,151.808
C05110=1100.880,111.218,-60.660,177.102,15.156,151.809
C05111=1100.874,110.969,-60.640,177.099,15.155,151.810
C05112=1100.869,110.720,-60.622,177.096,15.156,151.810
C05113=1100.863,110.470,-60.603,177.093,15.155,151.811
C05114=1100.858,110.221,-60.584,177.090,15.156,151.812
C05115=1100.852,109.972,-60.566,177.087,15.155,151.812
C05116=1100.846,109.723,-60.547,177.084,15.156,151.813
C05117=1100.840,109.473,-60.527,177.081,15.155,151.814
C05118=1100.834,109.224,-60.510,177.078,15.156,151.814
C05119=1100.829,108.975,-60.491,177.075,15.156,151.815
C05120=1100.823,108.725,-60.471,177.072,15.156,151.816
C05121=1100.817,108.476,-60.453,177.069,15.156,151.816
C05122=1100.812,108.228,-60.434,177.066,15.156,151.817
C05123=1100.807,107.978,-60.415,177.063,15.155,151.818
C05124=1100.800,107.728,-60.397,177.060,15.156,151.818
C05125=1100.795,107.480,-60.378,177.057,15.155,151.819
C05126=1100.789,107.230,-60.360,177.054,15.155,151.819
C05127=1100.784,106.981,-60.341,177.051,15.155,151.820
C05128=1100.778,106.732,-60.322,177.048,15.156,151.821
C05129=1100.772,106.483,-60.303,177.045,15.155,151.821
C05130=1100.767,106.233,-60.285,177.042,15.156,151.822
C05131=1100.761,105.984,-60.266,177.039,15.155,151.823
C05132=1100.755,105.735,-60.247,177.037,15.155,151.823
C05133=1100.750,105.485,-60.229,177.033,15.155,151.824
C05134=1100.744,105.236,-60.210,177.030,15.155,151.825
C05135=1100.739,104.987,-60.192,177.027,15.155,151.825
C05136=1100.732,104.738,-60.173,177.025,15.155,151.826
C05137=1100.727,104.488,-60.154,177.021,15.155,151.826
C05138=1100.721,104.239,-60.137,177.019,15.155,151.827
C05139=1100.716,103.990,-60.117,177.015,15.155,151.828
C05140=1100.711,103.741,-60.099,177.013,15.155,151.828
C05141=1100.704,103.491,-60.081,177.010,15.154,151.829
C05142=1100.699,103.243,-60.062,177.007,15.154,151.829
C05143=1100.693,102.993,-60.044,177.004,15.154,151.830
C05144=1100.688,102.744,-60.025,177.001,15.154,151.831
C05145=1100.682,102.495,-60.007,176.998,15.154,151.831
C05146=1100.676,102.245,-59.988,176.995,15.154,151.832
C05147=1100.671,101.996,-59.970,176.993,15.154,151.832
C05148=1100.665,101.747,-59.951,176.989,15.154,151.833
C05149=1100.659,101.498,-59.933,176.987,15.154,151.834
C05150=1100.654,101.248,-59.914,176.984,15.153,151.834
C05151=1100.648,100.999,-59.897,176.981,15.154,151.835
C05152=1100.643,100.750,-59.877,176.978,15.154,151.836
C05153=1100.637,100.501,-59.860,176.975,15.154,151.836
C05154=1100.631,100.251,-59.842,176.972,15.153,151.837
C05155=1100.626,100.002,-59.823,176.969,15.153,151.837
C05156=1100.620,99.752,-59.805,176.966,15.153,151.838
C05157=1100.613,99.503,-59.786,176.963,15.153,151.839
C05158=1100.609,99.254,-59.768,176.960,15.153,151.839
C05159=1100.602,99.005,-59.750,176.957,15.153,151.840
C05160=1100.597,98.756,-59.732,176.954,15.153,151.840
C05161=1100.591,98.506,-59.713,176.952,15.153,151.841
C05162=1100.585,98.257,-59.695,176.948,15.152,151.842
C05163=1100.579,98.008,-59.677,176.946,15.152,151.842
C05164=1100.574,97.758,-59.659,176.943,15.152,151.843
C05165=1100.568,97.509,-59.640,176.940,15.152,151.843
C05166=1100.563,97.260,-59.623,176.938,15.152,151.844
C05167=1100.557,97.010,-59.604,176.934,15.152,151.844
C05168=1100.551,96.762,-59.586,176.932,15.152,151.845
C05169=1100.545,96.512,-59.568,176.929,15.151,151.846
C05170=1100.540,96.239,-59.548,176.925,15.151,151.846
C05171=1100.533,95.966,-59.529,176.923,15.151,151.847
C05172=1100.527,95.692,-59.508,176.919,15.151,151.848
C05173=1100.521,95.420,-59.489,176.916,15.151,151.848
C05174=1100.515,95.170,-59.471,176.913,15.151,151.849
C05175=1100.510,94.921,-59.453,176.910,15.150,151.849
C05176=1100.504,94.672,-59.434,176.908,15.150,151.850
C05177=1100.498,94.423,-59.416,176.905,15.150,151.850
C05178=1100.492,94.173,-59.399,176.902,15.150,151.851
C05179=1100.487,93.923,-59.380,176.899,15.150,151.852
C05180=1100.482,93.674,-59.363,176.896,15.150,151.852
C05181=1100.475,93.425,-59.344,176.894,15.150,151.853
C05182=1100.470,93.176,-59.327,176.890,15.149,151.853
C05183=1100.465,92.927,-59.308,176.888,15.149,151.854
C05184=1100.459,92.677,-59.290,176.885,15.149,151.855
C05185=1100.453,92.428,-59.273,176.882,15.149,151.855
C05186=1100.447,92.178,-59.255,176.879,15.149,151.856
C05187=1100.442,91.929,-59.237,176.877,15.148,151.856
C05188=1100.436,91.681,-59.219,176.873,15.148,151.857
C05189=1100.430,91.431,-59.201,176.871,15.148,151.857
C05190=1100.425,91.182,-59.183,176.868,15.148,151.858
C05191=1100.419,90.933,-59.165,176.865,15.148,151.858
C05192=1100.413,90.683,-59.148,176.863,15.148,151.859
C05193=1100.408,90.434,-59.130,176.859,15.147,151.860
C05194=1100.402,90.184,-59.111,176.857,15.147,151.860
C05195=1100.397,89.935,-59.094,176.854,15.147,151.861
C05196=1100.391,89.686,-59.076,176.851,15.147,151.861
C05197=1100.385,89.436,-59.058,176.848,15.146,151.862
C05198=1100.380,89.187,-59.041,176.846,15.146,151.862
C05199=1100.374,88.937,-59.023,176.842,15.146,151.863
C05200=1100.368,88.688,-59.005,176.840,15.146,151.864
C05201=1100.362,88.439,-58.988,176.838,15.146,151.864
C05202=1100.356,88.189,-58.970,176.834,15.145,151.865
C05203=1100.351,87.940,-58.952,176.832,15.145,151.865
C05204=1100.345,87.691,-58.935,176.829,15.145,151.866
C05205=1100.339,87.442,-58.917,176.826,15.145,151.866
C05206=1100.334,87.193,-58.899,176.823,15.144,151.867
C05207=1100.328,86.943,-58.881,176.821,15.144,151.867
C05208=1100.322,86.694,-58.864,176.818,15.144,151.868
C05209=1100.317,86.445,-58.846,176.815,15.144,151.868
C05210=1100.311,86.196,-58.829,176.813,15.144,151.869
C05211=1100.305,85.946,-58.811,176.809,15.143,151.869
C05212=1100.299,85.697,-58.793,176.807,15.143,151.870
C05213=1100.294,85.448,-58.775,176.804,15.143,151.871
C05214=1100.288,85.198,-58.758,176.802,15.143,151.871
C05215=1100.283,84.949,-58.741,176.798,15.142,151.872
C05216=1100.277,84.700,-58.723,176.796,15.142,151.872
C05217=1100.271,84.450,-58.705,176.794,15.142,151.873
C05218=1100.265,84.201,-58.688,176.790,15.141,151.873
C05219=1100.260,83.952,-58.670,176.788,15.142,151.874
C05220=1100.254,83.703,-58.653,176.785,15.141,151.874
C05221=1100.248,83.452,-58.635,176.782,15.141,151.875
C05222=1100.242,83.204,-58.618,176.779,15.140,151.875
C05223=1100.237,82.955,-58.601,176.777,15.140,151.876
C05224=1100.231,82.705,-58.583,176.774,15.140,151.876
C05225=1100.225,82.456,-58.565,176.771,15.140,151.877
C05226=1100.220,82.206,-58.548,176.769,15.139,151.877
C05227=1100.214,81.957,-58.531,176.766,15.139,151.878
C05228=1100.209,81.708,-58.513,176.763,15.139,151.878
C05229=1100.203,81.458,-58.495,176.760,15.138,151.879
C05230=1100.197,81.209,-58.478,176.758,15.138,151.880
C05231=1100.192,80.960,-58.461,176.755,15.137,151.880
C05232=1100.186,80.711,-58.443,176.752,15.138,151.881
C05233=1100.181,80.461,-58.426,176.750,15.137,151.881
C05234=1100.175,80.188,-58.408,176.747,15.137,151.882
C05235=1100.168,79.914,-58.388,176.743,15.136,151.882
C05236=1100.161,79.642,-58.369,176.741,15.136,151.883
C05237=1100.155,79.368,-58.350,176.738,15.136,151.883
C05238=1100.150,79.119,-58.334,176.735,15.135,151.884
C05239=1100.145,78.870,-58.316,176.733,15.135,151.884
C05240=1100.139,78.621,-58.298,176.730,15.135,151.885
C05241=1100.134,78.371,-58.282,176.727,15.134,151.885
C05242=1100.127,78.122,-58.264,176.725,15.134,151.886
C05243=1100.122,77.872,-58.247,176.721,15.134,151.886
C05244=1100.116,77.623,-58.230,176.719,15.133,151.887
C05245=1100.111,77.374,-58.212,176.717,15.134,151.887
C05246=1100.105,77.125,-58.196,176.714,15.133,151.888
C05247=1100.099,76.875,-58.178,176.711,15.133,151.888
C05248=1100.093,76.625,-58.161,176.708,15.132,151.889
C05249=1100.088,76.376,-58.144,176.706,15.132,151.889
C05250=1100.082,76.127,-58.127,176.703,15.131,151.890
C05251=1100.076,75.878,-58.110,176.700,15.131,151.890
C05252=1100.071,75.629,-58.092,176.698,15.131,151.891
C05253=1100.064,75.379,-58.076,176.695,15.130,151.891
C05254=1100.059,75.130,-58.058,176.693,15.130,151.892
C05255=1100.054,74.880,-58.041,176.690,15.129,151.892
C05256=1100.047,74.631,-58.024,176.687,15.129,151.893
C05257=1100.042,74.382,-58.007,176.685,15.129,151.893
C05258=1100.037,74.132,-57.990,176.682,15.129,151.894
C05259=1100.031,73.883,-57.974,176.680,15.128,151.894
C05260=1100.025,73.633,-57.956,176.676,15.128,151.895
C05261=1100.019,73.384,-57.939,176.674,15.128,151.895
C05262=1100.013,73.134,-57.922,176.671,15.127,151.896
C05263=1100.008,72.885,-57.905,176.669,15.127,151.896
C05264=1100.003,72.636,-57.888,176.666,15.127,151.897
C05265=1099.996,72.387,-57.871,176.663,15.126,151.897
C05266=1099.991,72.137,-57.854,176.661,15.126,151.898
C05267=1099.985,71.888,-57.838,176.658,15.125,151.898
C05268=1099.980,71.639,-57.820,176.655,15.125,151.899
C05269=1099.975,71.389,-57.804,176.653,15.125,151.899
C05270=1099.968,71.140,-57.786,176.650,15.124,151.900
C05271=1099.962,70.890,-57.769,176.648,15.124,151.900
C05272=1099.956,70.641,-57.753,176.645,15.123,151.901
C05273=1099.951,70.392,-57.736,176.643,15.123,151.901
C05274=1099.946,70.142,-57.719,176.640,15.123,151.902
C05275=1099.940,69.893,-57.702,176.637,15.122,151.902
C05276=1099.934,69.644,-57.685,176.635,15.122,151.902
C05277=1099.928,69.394,-57.669,176.632,15.121,151.903
C05278=1099.923,69.145,-57.652,176.630,15.121,151.903
C05279=1099.917,68.895,-57.636,176.627,15.121,151.904
C05280=1099.912,68.646,-57.618,176.624,15.120,151.904
C05281=1099.906,68.397,-57.602,176.622,15.120,151.905
C05282=1099.900,68.147,-57.585,176.619,15.119,151.905
C05283=1099.895,67.898,-57.569,176.617,15.119,151.906
C05284=1099.889,67.649,-57.551,176.615,15.118,151.906
C05285=1099.883,67.400,-57.535,176.611,15.118,151.907
C05286=1099.878,67.150,-57.518,176.609,15.118,151.907
C05287=1099.871,66.900,-57.501,176.606,15.117,151.908
C05288=1099.865,66.651,-57.484,176.604,15.117,151.908
C05289=1099.860,66.401,-57.467,176.601,15.117,151.909
C05290=1099.854,66.152,-57.451,176.599,15.116,151.909
C05291=1099.849,65.902,-57.434,176.596,15.115,151.909
C05292=1099.843,65.653,-57.418,176.593,15.114,151.910
C05293=1099.837,65.404,-57.401,176.591,15.115,151.910
C05294=1099.831,65.155,-57.384,176.589,15.114,151.911
C05295=1099.825,64.905,-57.368,176.586,15.113,151.911
C05296=1099.820,64.656,-57.351,176.584,15.113,151.912
C05297=1099.814,64.406,-57.335,176.581,15.113,151.912
C05298=1099.808,64.133,-57.316,176.578,15.112,151.913
C05299=1099.802,63.860,-57.299,176.575,15.111,151.913
C05300=1099.796,63.587,-57.281,176.573,15.112,151.914
C05301=1099.789,63.314,-57.263,176.570,15.111,151.914
C05302=1099.784,63.064,-57.246,176.567,15.111,151.915
C05303=1099.778,62.815,-57.230,176.564,15.110,151.915
C05304=1099.772,62.566,-57.213,176.562,15.110,151.916
C05305=1099.766,62.316,-57.197,176.560,15.109,151.916
C05306=1099.761,62.067,-57.180,176.557,15.108,151.916
C05307=1099.755,61.817,-57.164,176.554,15.109,151.917
C05308=1099.749,61.568,-57.148,176.552,15.108,151.917
C05309=1099.743,61.319,-57.132,176.549,15.107,151.918
C05310=1099.737,61.069,-57.115,176.547,15.107,151.918
C05311=1099.732,60.820,-57.098,176.544,15.106,151.919
C05312=1099.726,60.570,-57.082,176.542,15.106,151.919
C05313=1099.720,60.321,-57.066,176.539,15.106,151.920
C05314=1099.714,60.072,-57.050,176.536,15.105,151.920
C05315=1099.708,59.822,-57.033,176.534,15.105,151.921
C05316=1099.702,59.573,-57.017,176.532,15.105,151.921
C05317=1099.697,59.323,-57.000,176.529,15.104,151.921
C05318=1099.691,59.074,-56.984,176.527,15.103,151.922
C05319=1099.685,58.825,-56.968,176.524,15.102,151.922
C05320=1099.679,58.575,-56.951,176.522,15.102,151.923
C05321=1099.673,58.326,-56.935,176.520,15.102,151.923
C05322=1099.668,58.076,-56.918,176.516,15.101,151.924
C05323=1099.662,57.827,-56.902,176.514,15.101,151.924
C05324=1099.656,57.578,-56.886,176.512,15.101,151.925
C05325=1099.650,57.328,-56.870,176.509,15.100,151.925
C05326=1099.645,57.079,-56.853,176.507,15.100,151.925
C05327=1099.639,56.829,-56.838,176.505,15.099,151.926
C05328=1099.633,56.580,-56.821,176.502,15.098,151.926
C05329=1099.628,56.331,-56.805,176.499,15.098,151.927
C05330=1099.622,56.081,-56.789,176.496,15.097,151.927
C05331=1099.616,55.832,-56.773,176.494,15.097,151.928
C05332=1099.610,55.583,-56.756,176.492,15.097,151.928
C05333=1099.605,55.332,-56.740,176.489,15.096,151.928
C05334=1099.599,55.084,-56.724,176.487,15.095,151.929
C05335=1099.593,54.834,-56.708,176.485,15.095,151.929
C05336=1099.587,54.585,-56.692,176.482,15.094,151.930
C05337=1099.582,54.336,-56.676,176.480,15.094,151.930
C05338=1099.576,54.086,-56.660,176.477,15.094,151.930
C05339=1099.570,53.836,-56.644,176.474,15.093,151.931
C05340=1099.564,53.587,-56.628,176.472,15.092,151.931
C05341=1099.559,53.338,-56.612,176.470,15.092,151.932
C05342=1099.553,53.088,-56.596,176.467,15.091,151.932
C05343=1099.548,52.839,-56.579,176.465,15.090,151.932
C05344=1099.542,52.589,-56.563,176.462,15.090,151.933
C05345=1099.536,52.339,-56.547,176.460,15.089,151.933
C05346=1099.531,52.091,-56.532,176.458,15.089,151.934
C05347=1099.525,51.841,-56.515,176.455,15.088,151.934
C05348=1099.519,51.591,-56.500,176.453,15.088,151.935
C05349=1099.513,51.342,-56.484,176.450,15.087,151.935
C05350=1099.507,51.093,-56.467,176.448,15.087,151.935
C05351=1099.502,50.843,-56.452,176.445,15.086,151.936
C05352=1099.496,50.594,-56.436,176.443,15.085,151.936
C05353=1099.490,50.345,-56.420,176.441,15.085,151.937
C05354=1099.485,50.095,-56.404,176.438,15.084,151.937
C05355=1099.479,49.846,-56.388,176.436,15.084,151.937
C05356=1099.473,49.597,-56.372,176.433,15.083,151.938
C05357=1099.468,49.347,-56.356,176.431,15.083,151.938
C05358=1099.462,49.097,-56.340,176.429,15.082,151.938
C05359=1099.457,48.848,-56.325,176.426,15.081,151.939
C05360=1099.451,48.599,-56.309,176.424,15.081,151.939
C05361=1099.445,48.349,-56.293,176.422,15.081,151.940
C05362=1099.439,48.075,-56.276,176.419,15.080,151.940
C05363=1099.434,47.802,-56.258,176.416,15.079,151.941
C05364=1099.427,47.529,-56.240,176.414,15.078,151.941
C05365=1099.421,47.255,-56.223,176.411,15.078,151.941
C05366=1099.415,47.006,-56.207,176.409,15.077,151.942
C05367=1099.410,46.756,-56.192,176.407,15.077,151.942
C05368=1099.404,46.507,-56.176,176.404,15.076,151.943
C05369=1099.398,46.257,-56.160,176.401,15.075,151.943
C05370=1099.393,46.008,-56.144,176.400,15.075,151.943
C05371=1099.387,45.758,-56.129,176.397,15.074,151.944
C05372=1099.381,45.509,-56.112,176.394,15.073,151.944
C05373=1099.375,45.260,-56.098,176.392,15.073,151.945
C05374=1099.370,45.011,-56.081,176.390,15.072,151.945
C05375=1099.364,44.761,-56.066,176.387,15.071,151.945
C05376=1099.359,44.512,-56.050,176.385,15.071,151.946
C05377=1099.353,44.262,-56.034,176.383,15.070,151.946
C05378=1099.348,44.013,-56.019,176.380,15.069,151.946
C05379=1099.342,43.763,-56.003,176.378,15.069,151.947
C05380=1099.336,43.513,-55.988,176.375,15.068,151.947
C05381=1099.330,43.264,-55.971,176.373,15.068,151.947
C05382=1099.325,43.015,-55.956,176.371,15.067,151.948
C05383=1099.319,42.765,-55.941,176.368,15.066,151.948
C05384=1099.313,42.516,-55.925,176.366,15.066,151.949
C05385=1099.308,42.266,-55.910,176.364,15.065,151.949
C05386=1099.302,42.017,-55.894,176.361,15.064,151.949
C05387=1099.296,41.767,-55.878,176.359,15.064,151.950
C05388=1099.291,41.518,-55.863,176.357,15.063,151.950
C05389=1099.285,41.268,-55.848,176.354,15.062,151.951
C05390=1099.279,41.019,-55.832,176.352,15.062,151.951
C05391=1099.274,40.770,-55.816,176.350,15.061,151.951
C05392=1099.267,40.520,-55.801,176.347,15.061,151.952
C05393=1099.262,40.271,-55.786,176.345,15.060,151.952
C05394=1099.256,40.021,-55.770,176.343,15.059,151.952
C05395=1099.251,39.771,-55.754,176.340,15.059,151.953
C05396=1099.245,39.522,-55.740,176.338,15.058,151.953
C05397=1099.239,39.273,-55.724,176.336,15.058,151.953
C05398=1099.233,39.023,-55.708,176.333,15.057,151.954
C05399=1099.228,38.774,-55.693,176.331,15.056,151.954
C05400=1099.222,38.524,-55.678,176.329,15.056,151.955
C05401=1099.217,38.276,-55.662,176.327,15.055,151.955
C05402=1099.211,38.026,-55.647,176.324,15.054,151.955
C05403=1099.205,37.776,-55.632,176.322,15.054,151.956
C05404=1099.200,37.527,-55.616,176.320,15.053,151.956
C05405=1099.194,37.277,-55.600,176.317,15.052,151.956
C05406=1099.187,37.028,-55.585,176.315,15.052,151.957
C05407=1099.182,36.778,-55.570,176.313,15.051,151.957
C05408=1099.176,36.529,-55.555,176.310,15.050,151.957
C05409=1099.171,36.279,-55.540,176.308,15.050,151.958
C05410=1099.165,36.029,-55.524,176.306,15.050,151.958
C05411=1099.158,35.780,-55.509,176.304,15.049,151.959
C05412=1099.153,35.531,-55.494,176.301,15.048,151.959
C05413=1099.147,35.282,-55.479,176.299,15.047,151.959
C05414=1099.142,35.032,-55.463,176.297,15.047,151.960
C05415=1099.136,34.783,-55.448,176.294,15.046,151.960
C05416=1099.130,34.533,-55.433,176.292,15.045,151.960
C05417=1099.125,34.283,-55.418,176.290,15.045,151.961
C05418=1099.119,34.034,-55.403,176.287,15.044,151.961
C05419=1099.113,33.785,-55.387,176.285,15.043,151.961
C05420=1099.107,33.535,-55.372,176.283,15.043,151.962
C05421=1099.102,33.286,-55.357,176.281,15.042,151.962
C05422=1099.095,33.036,-55.342,176.278,15.041,151.963
C05423=1099.090,32.787,-55.327,176.276,15.041,151.963
C05424=1099.084,32.538,-55.312,176.274,15.040,151.963
C05425=1099.078,32.288,-55.296,176.271,15.039,151.964
C05426=1099.072,32.015,-55.280,176.269,15.039,151.964
C05427=1099.066,31.741,-55.264,176.266,15.038,151.964
C05428=1099.060,31.467,-55.247,176.264,15.037,151.965
C05429=1099.054,31.195,-55.230,176.261,15.036,151.965
C05430=1099.048,30.945,-55.215,176.259,15.035,151.965
C05431=1099.042,30.696,-55.200,176.257,15.035,151.966
C05432=1099.037,30.445,-55.185,176.255,15.034,151.966
C05433=1099.031,30.196,-55.171,176.252,15.033,151.966
C05434=1099.025,29.946,-55.155,176.250,15.033,151.967
C05435=1099.020,29.697,-55.141,176.248,15.032,151.967
C05436=1099.014,29.447,-55.125,176.246,15.032,151.967
C05437=1099.008,29.198,-55.110,176.243,15.031,151.968
C05438=1099.002,28.949,-55.095,176.241,15.030,151.968
C05439=1098.997,28.699,-55.080,176.239,15.030,151.969
C05440=1098.990,28.450,-55.065,176.237,15.028,151.969
C05441=1098.985,28.200,-55.050,176.234,15.028,151.969
